//     PlcTask Outputs/Output.Out_Moter_Error <-> PlcTask Inputs/ExpConver.Out_Moter_Error
//     PlcTask Outputs/Output.Out_Moter_Running <-> PlcTask Inputs/ExpConver.Out_Moter_Running
//     PlcTask Outputs/Output.Out_Pos_sensor <-> PlcTask Inputs/ExpConver.Out_sensor
//     PlcTask Outputs/Output.PullOver_bBuzy <-> PlcTask Inputs/ExpConver.PullOver_bBuzy
//     PlcTask Outputs/Output.PullOver_bDone <-> PlcTask Inputs/ExpConver.PullOver_bDone
//     PlcTask Outputs/Output.PullOver_bError <-> PlcTask Inputs/ExpConver.PullOver_bError
//     PlcTask Outputs/Output.in_Pos_sensor <-> PlcTask Inputs/ExpConver.In_sensor

CONFIGURATION Main
    RESOURCE PLC ON TwinCAT3
        TASK PlcTask(INTERVAL := T#10ms, PRIORITY := 14);
        PROGRAM MAIN WITH PlcTask : MAIN;
    END_RESOURCE
END_CONFIGURATION

// ---- DUTs/ActionMode.TcDUT
{attribute 'qualified_only'}
{attribute 'strict'}
TYPE ActionMode :
(
	DoNothing	:= 0,
	AbsMove		:= 1,
	RelMove		:= 2,
	Home		:= 3,
	Find		:= 4
);
END_TYPE

// ---- DUTs/IO模組/IO_In16.TcDUT
TYPE IO_In16 :
STRUCT
	in AT %I* : ARRAY [1..16] OF BOOL;
END_STRUCT
END_TYPE

// ---- DUTs/IO模組/IO_Out16.TcDUT
TYPE IO_Out16 :
STRUCT
	Out AT %Q* : ARRAY [1..16] OF BOOL;
END_STRUCT
END_TYPE

// ---- DUTs/Jog_STRUCT/Jog_Laser_Group.TcDUT
TYPE Jog_Laser_Group :
STRUCT
	// 位置	
	Pos : XYZ_Point;
	
	// Jog模式 X軸 前進
	X_P_S : BOOL;
	// Jog模式 X軸 後退
	X_N_S : BOOL;
	
	// Jog模式 Y軸 前進
	Y_P_S : BOOL;
	// Jog模式 Y軸 後退
	Y_N_S : BOOL;
	
	// Jog模式 Z軸 前進
	Z_P_S : BOOL;
	// Jog模式 Z軸 後退
	Z_N_S : BOOL;

	// Jog模式 X軸 前進
	X_P : BOOL;
	// Jog模式 X軸 後退
	X_N : BOOL;
	
	// Jog模式 Y軸 前進
	Y_P : BOOL;
	// Jog模式 Y軸 後退
	Y_N : BOOL;
	
	// Jog模式 Z軸 前進
	Z_P : BOOL;
	// Jog模式 Z軸 後退
	Z_N : BOOL;
	
	
	// 雷射吹氣_狀態
	Laser_Blow_s : BOOL;
	// 雷射護蓋_狀態
	Laser_Cover_s : BOOL;
	

	// 雷射吹氣
	Laser_Blow : BOOL;
	// 雷射護蓋
	Laser_Cover : BOOL;
END_STRUCT
END_TYPE

// ---- DUTs/Jog_STRUCT/Jog_Fx_Group.TcDUT
TYPE Jog_Fx_Group :
STRUCT
	// 
	P_S : BOOL;
	// 後退
	N_S : BOOL;
	
	// 前進
	P : BOOL;
	// 後退
	N : BOOL;
	
	
	// 前進
	P_Fast_S : BOOL;
	// 後退
	N_Fast_S : BOOL;	

	// 前進
	P_Fast : BOOL;
	// 後退
	N_Fast : BOOL;
	
	
	// 下壓夾狀態
	V_Close_S : BOOL;
	// 下壓開狀態
	V_Open_S : BOOL;
	
	// 下壓夾
	V_Close : BOOL;
	// 下壓開
	V_Open : BOOL;
	
	// 滾輪夾狀態
	H_Close_S : BOOL;
	// 滾輪開狀態
	H_Open_S : BOOL;
	// 滾輪夾保持狀態
	H_Hold_S : BOOL;
	
	// 滾輪夾
	H_Close : BOOL;
	// 滾輪開
	H_Open : BOOL;
	// 滾輪夾保持
	H_Hold : BOOL;
	
	// 外部編碼器接觸
	ExEncTouch : BOOL;
	// 外部編碼器脫離
	ExEncExit : BOOL;
END_STRUCT
END_TYPE

// ---- DUTs/MachineState.TcDUT
{attribute 'qualified_only'}
{attribute 'strict'}
TYPE MachineState :
(
	standby := 0, 			// 待命
	Auto_mode := 2#01,		// 自動模式
	auto_mode_wait := 2#10,		// 自動模式等待中
	Remote_Auto_mode := 2#11,		// 遠端自動模式
	manual_mode := 2#100,	// 手動模式
	Homing_mode := 2#1000,		// 歸零模式
	
	error := 16#20,	// 發生錯誤
	Door := 16#40,		// 安全光柵觸發
	emergency := 16#80	// 緊急停止
) INT;
END_TYPE

// ---- DUTs/Sub_Step.TcDUT
TYPE Sub_Step :
STRUCT
	Step	: INT;
	
	bBuzy	: BOOL;
	bDone	: BOOL;
	bError	: BOOL;
END_STRUCT
END_TYPE

// ---- DUTs/TestAction.TcDUT
TYPE TestAction :
STRUCT
	// 選擇的動作 (1.軸移動、 2.等待完成、 3.等待時間 、4. 重複)
	ActionSelect: INT;
	
	// 選擇的軸 (動作1 有效)
	AxisSelect: INT;
	
	// 移動位置 (動作1 有效)
	Pos : REAL;
	
	// 移動速度 (動作1 有效)
	Speed: REAL;
	
	// 等待時間(動作3 有效)
	WaitTime : REAL;
	
	// 重複次數(動作4 有效)
	Cycles: UINT;
	
	// 重複動作(動作4 有效)
	Cycles_StartStep: UINT;
	
	// 重複次數(動作4 有效)
	Cycles_Done: UINT;
END_STRUCT
END_TYPE

// ---- DUTs/加工資料結構/材料加工資訊結構/tsSteelData.TcDUT
// 專案資料結構
TYPE tsSteelData :
STRUCT
	// 素材編號 (uuid)
	uid							: STRING(36);
	// 型鋼類型
	SteelType					: DINT;
	// 長度
	Length						: LREAL;
	// 高度
	Height						: LREAL;
	// 寬度
	Width						: LREAL;
	// 翼板厚度t1
	T1							: LREAL;
	// 翼板厚度t2
	T2							: LREAL;
	// 原點偏移
	OriginOffset				: LREAL;
	// 開啟預覽
	PreviewEnabled				: BOOL;
	// 預覽模式
	PreviewMode					: DINT;
	// 預覽時間
	PreviewTme					: DINT;
	// 「指定區域加工模式」的起始範圍
	rDesignateAreaRangeBegin	: LREAL;
	// 「指定區域加工模式」的結束範圍
	rDesignateAreaRangeEnd		: LREAL;
	
	// 上面的加工內容
	payloadTop					: STRING(36);
	// 下面的加工內容
	payloadBottom				: STRING(36);
	// 左面的加工內容
	payloadLeft					: STRING(36);
	// 右面的加工內容
	payloadRight				: STRING(36);
	
	// 全部加工完成
	bJobFinish					:BOOL;
END_STRUCT
END_TYPE

// ---- DUTs/加工資料結構/工單結構/WorkOrder_Data.TcDUT
// 專案資料結構
TYPE WorkOrder_Data :
STRUCT
	// 加工順序
	SN			: DINT;
	// 高
	Height		: LREAL;
	// 寬
	Width		: LREAL;
	// 素材編號 (uuid)
	steel_id	: STRING(36);
END_STRUCT
END_TYPE

// ---- DUTs/加工資料結構/雷射加工參數/LaserParameter_Data.TcDUT
TYPE LaserParameter_Data :
STRUCT
	// 加工參數代碼
	id				: DINT;
	// 螺徑(mm)
	SpiralDiameter	: LREAL;
	// 螺距(mm)
	SpiralDist		: LREAL;
	// 功率(%)
	Power			: DINT;
	// 速度(mm/S)
	Speed			: DINT;	
	// 頻率(KHZ)
	FREQ			: DINT;	
	// 脈波寬度(ns)
	PulseWidth		: DINT;	
END_STRUCT
END_TYPE

// ---- DUTs/加工資料結構/雷射加工資料/LaserProcess_Data.TcDUT
TYPE LaserProcess_Data :
// 115 byte
STRUCT
	// 資料的UID
	data_uid					: STRING(36);
	// 面的UID
	uid							: STRING(36);
	// 該面的序號(順序)
	paySerial					: DINT;
	// 使用雷射參數
	LaserParameter				: DINT;
	// 加工內容的x座標
	Point_X						: LREAL;
	// 加工內容的y座標
	Point_Y						: LREAL;
	// 加工內容的寬度
	Width						: LREAL;
	// 加工內容的高度
	Height						: LREAL;
	// 是否是QRCode
	isQRCode					: BOOL;
	// 已完成
	isDone						: BOOL;
	// QRCode字串
	qrcode_data					: STRING(100);
END_STRUCT
END_TYPE

// ---- DUTs/座標/XYZ_Point.TcDUT
TYPE XYZ_Point :
STRUCT
	X : LREAL;
	Y : LREAL;
	Z : LREAL;
END_STRUCT
END_TYPE

// ---- MSG/訊息格式/MsgLevel.TcDUT
{attribute 'qualified_only'}
{attribute 'strict'}
TYPE MsgLevel :
(
	Error	:= 4,
	Alarm	:= 2,
	Info	:= 1,
	None	:= 0
	
)INT;
END_TYPE

// ---- MSG/訊息格式/MsgStruct.TcDUT
{attribute 'pack_mode' := '1'} 
TYPE MsgStruct :
STRUCT
	// 訊息時間
	msgTIME		: DATE_AND_TIME;
	// 訊息等級
	Level		: MsgLevel;
	// 訊息號碼
	Number	: UINT;
	// 訊息附帶文字1
	MsgStr1	: WSTRING(80);
	// 訊息附帶文字2
	MsgStr2	: WSTRING(80);
	// 訊息全文
	raw_msg_str	: WSTRING(250);
END_STRUCT
END_TYPE

// ---- MSG/訊息格式/MsgStruct_RAW.TcDUT
{attribute 'pack_mode' := '1'} 
TYPE MsgStruct_RAW :
STRUCT
	// 訊息時間
	msgTIME		: DATE_AND_TIME;
	// 訊息等級
	Level		: MsgLevel;
	// 訊息號碼
	Number	: UINT;
	// 訊息附帶文字1
	MsgStr1	:  ARRAY[0..159] OF BYTE;
	// 訊息附帶文字2
	MsgStr2	: ARRAY[0..159] OF BYTE;
	// 訊息全文
	raw_msg_str	: ARRAY[0..499] OF BYTE;
END_STRUCT
END_TYPE

// ---- POUs/功能塊/資料庫 Postgre相關/相關結構/取得範圍內的加工資料/SQL_Get_Payload_Struct.TcDUT

TYPE SQL_Get_Payload_Struct :
STRUCT
	// 
	Payload_Uid : STRING(36);
	PosBegain	: LREAL;
	PosEnd	: LREAL;
END_STRUCT
END_TYPE

// ---- POUs/功能塊/資料庫 Postgre相關/相關結構/取得X點/SQL_GetPosX_Struct.TcDUT
// 取得檔案的參數
TYPE SQL_GetPosX_Struct :
STRUCT
	Payload_A_Uid : STRING(36);
	Payload_B_Uid : STRING(36);
	Payload_C_Uid : STRING(36);
	Payload_D_Uid : STRING(36);
	Pos	: LREAL;
END_STRUCT
END_TYPE

// ---- POUs/功能塊/資料庫 Postgre相關/相關結構/寫入起始時間/Payload_Write_Time.TcDUT
TYPE Payload_Write_Time :
STRUCT
	// 時間
	Start_TIME		: DATE_AND_TIME;
	// 目標uid
	Uid : STRING(36);
END_STRUCT
END_TYPE

// ---- POUs/功能塊/資料庫 Postgre相關/記錄用/程式紀錄/StepLog_Struct.TcDUT
TYPE StepLog_Struct :
STRUCT
	step_number : DINT;
	created_at : LINT;
	program_name : STRING(80);
	extras_Srt : STRING(255) := '{}';
END_STRUCT
END_TYPE

// ---- POUs/動作流程控制/測試功能/Sql_TestData.TcDUT
TYPE Sql_TestData :
STRUCT
	ID : LINT;
	LogTime : DATE_AND_TIME;
	
END_STRUCT
END_TYPE

// ---- POUs/動作流程控制/測試功能/Sql_TestWriteData.TcDUT
TYPE Sql_TestWriteData :
STRUCT
	LogTime : DATE_AND_TIME;
END_STRUCT
END_TYPE

// ---- GVLs/Axis.TcGVL
{attribute 'TcContextName':='PlcTask'}
VAR_GLOBAL
// 軸控制
// ============== 滾輪軸 ==============
	//  前
	Axis_FX1: AXIS_REF;
	//  後
	Axis_FX2: AXIS_REF;
	
	Fx : AxisFx;
	
	
// ============== A ==============
	
	// X軸
	Axis_AX: AXIS_REF;
	
	// Y軸
	Axis_AY: AXIS_REF;
	// Z軸
	Axis_AZ1: AXIS_REF;
	Axis_AZ2: AXIS_REF;
	
	GaX : AxisBase;
	GaY : AxisBase;
	GaZ : MultipleAxisBase;
	

	
// ============== B ==============
	// X軸
	Axis_BX: AXIS_REF;
	// Y軸
	Axis_BY1: AXIS_REF;
	Axis_BY2: AXIS_REF;
	// Z軸
	Axis_BZ: AXIS_REF;
	
	GbX : AxisBase;
	GbY : MultipleAxisBase;
	GbZ : AxisBase;
	
// ============== C ==============
	// X軸
	Axis_CX: AXIS_REF;
	// Y軸
	Axis_CY: AXIS_REF;
	// Z軸
	Axis_CZ1: AXIS_REF;
	Axis_CZ2: AXIS_REF;
	
	GcX : AxisBase;
	GcY : AxisBase;
	GcZ : MultipleAxisBase;
	
// ============== D ==============
	// X軸
	Axis_DX: AXIS_REF;
	// Y軸
	Axis_DY: AXIS_REF;
	// Z軸
	Axis_DZ: AXIS_REF;
	
	GdX : AxisBase;
	GdY : AxisBase;
	GdZ : AxisBase;


//  ============== 整體軸速度 ==============	
	Override: LREAL := 100;
	bIsHome: BOOL;
	bPower: BOOL;
	
{region "============= 編碼器  ============="}
	Encoder_FxA_PosEnc	:	MDP5001_511_5ED3066D;
	Encoder_FxB_PosEnc	:	MDP5001_511_5ED3066D;
		 
	Encoder_FxA_Clamp	:	MDP5001_511_5ED3066D;
	Encoder_FxB_Clamp	:	MDP5001_511_5ED3066D;
		 
	Encoder_FxA_ExPosEnc	:	MDP5001_511_5ED3066D;
	Encoder_FxB_ExPosEnc	:	MDP5001_511_5ED3066D;
	
	// FxA外部位置
	FxA_Exp_Pos				: LREAL;
	// FxB外部位置
	FxB_Exp_Pos				: LREAL;
	
	// Fx整合位置
	Fx_Exp_Pos				: LREAL;
{endregion}
	

	id: INT;
	
	
END_VAR


VAR_GLOBAL PERSISTENT
	// Gax軸 移動距離
	GaX_total_Move: LREAL;
	// Gay軸 移動距離
	GaY_total_Move: LREAL;
	// Gaz軸 移動距離
	GaZ_total_Move: LREAL;
	
	// Gax軸 移動距離
	GbX_total_Move: LREAL;
	// Gay軸 移動距離
	GbY_total_Move: LREAL;
	// Gaz軸 移動距離
	GbZ_total_Move: LREAL;
	
	// Gax軸 移動距離
	GcX_total_Move: LREAL;
	// Gay軸 移動距離
	GcY_total_Move: LREAL;
	// Gaz軸 移動距離
	GcZ_total_Move: LREAL;
	
	// Gax軸 移動距離
	GdX_total_Move: LREAL;
	// Gay軸 移動距離
	GdY_total_Move: LREAL;
	// Gaz軸 移動距離
	GdZ_total_Move: LREAL;
	
	// Gax軸 移動距離
	GaX_Last_Oil: LREAL;
	// Gay軸 移動距離
	GaY_Last_Oil: LREAL;
	// Gaz軸 移動距離
	GaZ_Last_Oil: LREAL;
	
	// Gax軸 移動距離
	GbX_Last_Oil: LREAL;
	// Gay軸 移動距離
	GbY_Last_Oil: LREAL;
	// Gaz軸 移動距離
	GbZ_Last_Oil: LREAL;
	
	// Gax軸 移動距離
	GcX_Last_Oil: LREAL;
	// Gay軸 移動距離
	GcY_Last_Oil: LREAL;
	// Gaz軸 移動距離
	GcZ_Last_Oil: LREAL;
	
	// Gax軸 移動距離
	GdX_Last_Oil: LREAL;
	// Gay軸 移動距離
	GdY_Last_Oil: LREAL;
	// Gaz軸 移動距離
	GdZ_Last_Oil: LREAL;
END_VAR

// ---- GVLs/GrobelVariable.TcGVL
VAR_GLOBAL
// 雜項
	
	ProgramReset:BOOL;
	
	// 機器已回零
	bHome : BOOL;
	
	// 
	LogFx : FxErrPos;
END_VAR

VAR_GLOBAL PERSISTENT
	// 運轉次數
	uRunCounter:UDINT;
END_VAR

// ---- GVLs/Hmi.TcGVL
{attribute 'qualified_only'}
VAR_GLOBAL
(* ================= 模式選擇 ================= *)
	// 自動模式
	Auto_Mode : BOOL;

	// Jog模式
	Jog_Mode : BOOL;
	
	// 手輪模式
	MPG_Mode : BOOL;
	
	// 選擇的模式
	Mode_Select : DINT;

(* ================= 自動模式 ================= *)
	// 自動流程 開始執行
	Auto_Start : BOOL;
	
	// 一循環流程 開始執行
	Auto_OneCycle_Start : BOOL;
	
	// 自動流程 暫停/繼續
	Auto_Pause:BOOL;
	
	// 自動流程 加工單
	Auto_ProjectWorkOrder_uuid : STRING;

	// 自動流程 動作選擇
	Auto_ProgramSelect : DINT;

	// 自動流程 動作執行中
	Auto_bBuzy : BOOL;
	
	// 自動流程 動作完成
	Auto_bDone : BOOL;
	
	

	// 動作狀態通知
	ActinoNow:WSTRING;
	

	// 狀態欄 機器動作中
	State: MachineState := MACHINESTATE.standby;
	
	
(*==================== Jog模式====================*)
	// Jog模式 軸組選擇
	Jog_GroupSelect : DINT;
	
	// Jog模式 互鎖解除
	Jog_UnLimite : BOOL;
	
	// Jog模式 速度
	Jog_Speed: REAL := 30;
	
	
	
	Jog_move_to : LREAL;
	Jog_move_to_start : BOOL;
	Jog_move_to_bBuzy : BOOL;
	Jog_move_to_bDone : BOOL;
	
	// JOG 設定動作群組
	Jog_Set_GroupA: BOOL;
	Jog_Set_GroupB: BOOL;
	Jog_Set_GroupC: BOOL;
	Jog_Set_GroupD: BOOL;
	
	// Jog模式 X軸 前進
	Jog_X_P : BOOL;
	// Jog模式 X軸 後退
	Jog_X_N : BOOL;
	
	// Jog模式 Y軸 前進
	Jog_Y_P : BOOL;
	// Jog模式 Y軸 後退
	Jog_Y_N : BOOL;
	
	// Jog模式 Z軸 前進
	Jog_Z_P : BOOL;
	// Jog模式 Z軸 後退
	Jog_Z_N : BOOL;
	
	
(*==================== 原點設置 ====================*)
	// 設定 X軸 原點
	Set_X_Home : BOOL;
	// 設定 X軸 正極限
	Set_X_P_Limite : BOOL;
	// 設定 Y軸 原點
	Set_Y_Home : BOOL;
	// 設定 Y軸 正極限
	Set_Y_P_Limite : BOOL;
	// 設定 Z軸 原點
	Set_Z_Home : BOOL;
	// 設定 Z軸 正極限
	Set_Z_P_Limite : BOOL;

	
	
	// 將極限設定 參數 寫入軸
	Set_Axis_Limit : BOOL;
	
	// 錯誤重置
	SysErrorRest: BOOL;
	


	
	
END_VAR

// ---- GVLs/Hmi_Web.TcGVL
{attribute 'qualified_only'}
VAR_GLOBAL
(* ================= 模式選擇 ================= *)
	// 人機 > PLC WatchDog
	Watchdog_in : BOOL;
	
	// PLC > 人機 WatchDog
	Watchdog_Out : BOOL;
	
	// 錯誤重置
	SysErrorRest: BOOL;
	
	// 自動模式
	Auto_Mode : BOOL;
	
	// 單步模式
	Auto_Step_mode_Enable :BOOL;
	
	
	// 單步模式生效
	Auto_Step_active :BOOL;

	// Jog模式
	Jog_Mode : BOOL;
	
	// 手輪模式
	MPG_Mode : BOOL;
	
	// 選擇的模式
	Mode_Select : DINT;
	

(* ================= 自動模式 ================= *)
	// 自動流程 開始的專案UUID
	Auto_ProjectWorkOrder_uuid : STRING(36);
	// 自動流程 開始的專案UUID
	Start_WorkOrder_UUID : STRING(36);

	// 自動流程 開始執行
	Auto_Start : BOOL;
	
	Auto_OneCycle_Start : BOOL;
	
	
	
	

	
	// 自動流程 暫停/繼續
	Auto_Pause:BOOL;

	// 自動流程 動作選擇
	Auto_ProgramSelect : DINT;

	// 自動流程 動作執行中
	Auto_bBuzy : BOOL;
	
	// 自動流程 動作完成
	Auto_bDone : BOOL;
	
	// 自動流程 原點復歸
	Auto_homming : BOOL;
	
	// 動作狀態通知
	ActinoNow:WSTRING;
	
	// 狀態欄 機器動作中
	State: MachineState := MACHINESTATE.standby;
	
	
	// 雷射A 控制
	Process_Data_UUID_A				: STRING(36);
 	Process_Data_UUID_A_Start		: BOOL;
	// 雷射B 控制
	Process_Data_UUID_B				: STRING(36);
 	Process_Data_UUID_B_Start		: BOOL;
	// 雷射C 控制
	Process_Data_UUID_C				: STRING(36);
 	Process_Data_UUID_C_Start		: BOOL;
	// 雷射D 控制
	Process_Data_UUID_D				: STRING(36);
 	Process_Data_UUID_D_Start		: BOOL;
	
(*==================== Jog模式====================*)
	// Jog模式 軸組選擇
	Jog_GroupSelect : DINT;
	
	// Jog模式 互鎖解除
	Jog_UnLimite : BOOL;
	
	// Jog模式 速度
	Jog_Speed: REAL := 80;
	
	jog_trig_R : ARRAY [0..9] OF R_TRIG;


	jog_trig_F : ARRAY [0..9] OF F_TRIG; 
	
	
(*==================== Ga Jog模式====================*)	
	// Jog模式Ga X軸 前進
	Jog_Ga : Jog_Laser_Group;
	

(*==================== Gb Jog模式====================*)	
	// Jog模式Gb X軸 前進
	Jog_Gb : Jog_Laser_Group;

(*==================== Gc Jog模式====================*)	
	// Jog模式Gc
	Jog_Gc : Jog_Laser_Group;

(*==================== Gd Jog模式====================*)	
	// Jog模式Gd
	Jog_Gd : Jog_Laser_Group;
	
(*==================== FX A Jog模式====================*)	
	// Jog模式FxA
	Jog_FxA : Jog_Fx_Group;
	
(*==================== FX A Jog模式====================*)	
	// Jog模式FxB
	Jog_FxB : Jog_Fx_Group;
	
	// 油壓幫浦
	Oil_Pump:BOOL;
(*==================== Fx 目前位置====================*)	
	Fx_Pos			:LREAL;		// Fx 馬達位置
	FxA_Ex_Pos		:LREAL;		// FxA 測長盤
	FxB_Ex_Pos		:LREAL;		// FxB 測長盤

	FxA_H_Pos		:LREAL;		// FxA 油壓夾輪位置
	FxB_H_Pos		:LREAL;		// FxB 油壓夾輪位置
	
	
(*==================== Ga 工件座標系位置====================*)	
	WCS_A : XYZ_Point;
(*==================== Gb 工件座標系位置====================*)	
	WCS_B : XYZ_Point;
(*==================== Gc 工件座標系位置====================*)	
	WCS_C : XYZ_Point;
(*==================== Gd 工件座標系位置====================*)	
	WCS_D : XYZ_Point;
	
	
END_VAR
VAR_GLOBAL PERSISTENT
	// 工件誤差修正
	Auto_Steel_X_Offset : LREAL;
END_VAR

// ---- GVLs/MaCfg.TcGVL
{attribute 'qualified_only'}
VAR_GLOBAL PERSISTENT
	(* ======= Group A =======*)
	// 雷射頭A焦距
	laserA_Dis : REAL := 297;
	// 軸組A的 雷射測距可以測得範圍
	laserA_Y_DisSensorArrivePos	:REAL := 300;
	// 軸組Ax的 雷射測距點 到 雷射頭的中心點
	laserA_X_DisSensor2LaserCenter : REAL := -76;
	// 軸組Ay的 雷射測距點 到 雷射頭的中心點
	laserA_Y_DisSensor2LaserCenter : REAL := 12;
	// 軸組A的 Y 基準位置 (實際無法到達) (搭配 FindY 指令，可以測得工件高度)
	laserA_Y_ReferencePos : REAL := 677.7;
	
	(* ======= Group B =======*)
	// 雷射頭B焦距
	laserB_Dis	: REAL := 297;
	// 軸組B的 雷射測距可以測得範圍
	laserB_Y_DisSensorArrivePos		: REAL := 185;
	
	// 軸組Bx的 雷射測距點 到 雷射頭的中心點
	laserB_X_DisSensor2LaserCenter	: REAL := -0.6;
	// 軸組By的 雷射測距點 到 雷射頭的中心點
	laserB_Y_DisSensor2LaserCenter	: REAL := -77.2;
	
	// 軸組B的 Y 基準位置 (搭配 FindY 指令，可以測得工件高度)
	laserB_Y_ReferencePos	: REAL := 1344.5599;
	// 軸組B的 Z 基準位置 (實際無法到達)
	laserB_Z_ReferencePos	: REAL := -298;
	
	// 軸組Bx的 雷射測距點 到 雷射頭的中心點
	laserB_Y_safetyPos	: REAL := 20;
	// 軸組B的Z軸的安全位置
	laserB_Z_safetyPos		: REAL := 500;
	
	
	(* ======= Group C =======*)
	// 雷射頭C焦距
	laserC_Dis : REAL := 298;
	// 軸組C的 雷射測距可以測得範圍
	laserC_Y_DisSensorArrivePos	:REAL := 185;
	// 軸組Cx的 雷射測距點 到 雷射頭的中心點
	laserC_X_DisSensor2LaserCenter : REAL := 77.9;
	// 軸組Cy的 雷射測距點 到 雷射頭的中心點
	laserC_Y_DisSensor2LaserCenter : REAL := 5.8;
	// 軸組C的 Y 基準位置 (實際無法到達) (搭配 FindY 指令，可以測得工件高度)
	laserC_Y_ReferencePos : REAL := 605.3;
	// 軸組C的 Z 基準位置 (實際無法到達)
	laserC_Z_ReferencePos : REAL := -416;
	
	(* ======= Group D =======*)
	// 雷射頭D焦距
	laserD_Dis : REAL := 299;
	// 軸組D的 雷射測距可以測得範圍
	laserD_Y_DisSensorArrivePos	:REAL := 185;
	// 軸組D的 雷射測距點 到 雷射頭的中心點
	laserD_Y_DisSensor2LaserDenter : REAL := 3.1;
	// 軸組D的 Y 基準位置 (實際無法到達) (搭配 FindY 指令，可以測得工件高度)
	laserD_Y_ReferencePos : REAL := 1286.064821;
	
	
	// FxB被動編碼器 比例(mm/plus)
	FxA_Enc_Scale : LREAL := 0.046047445;
	// FxB測常盤編碼器 比例(mm/plus)
	FxA_Enc_Ext_Scale : LREAL := 0.14459929225;
	
	// FxB被動編碼器 比例(mm/plus)
	FxB_Enc_Scale : LREAL := 0.046047445;
	// FxB測常盤編碼器 比例(mm/plus)
	FxB_Enc_Ext_Scale : LREAL := 0.14459929225;
	
	
	
	// 進料端反轉
	bInSite_Invert: BOOL;
	
	//
	// AC夾輪的零點位置 ( 空夾位置 + 空夾兩夾輪間距(70))
	FxA_Clamp_Zero_Pos: LREAL := 1297.4;
	// BD夾輪的零點位置 ( 空夾位置 + 空夾兩夾輪間距(70))
	FxB_Clamp_Zero_Pos: LREAL := 1296.49;
	
	// 雷射動作超時
	LaserPrinter_Timeout : DINT := 60000;
	
END_VAR

// ---- GVLs/IO.TcGVL
{attribute 'qualified_only'}
{attribute 'TcContextName':='PlcTask'}
VAR_GLOBAL
{region "============= EL1409_1 ============="}
	// 緊急停止-PB
	i101 AT %I*: BOOL;
	// IPC開機-PB
	i102 AT %I*: BOOL;
	// 程式暫停-PB
	i103 AT %I*: BOOL;
	// 程式啟動-PB
	i104 AT %I*: BOOL;
	// 重置-PB
	i105 AT %I*: BOOL;
	// 原點模式A-KS
	i106 AT %I*: BOOL;
	// 原點模式B-KS
	i107 AT %I*: BOOL;
	// 吋動-KS
	i108 AT %I*: BOOL;
	// 半自動-KS
	i109 AT %I*: BOOL;
	// 全自動-KS
	i110 AT %I*: BOOL;
	// 門解鎖-KS
	i111 AT %I*: BOOL;
	// 安全模組重置-PB
	i112 AT %I*: BOOL;
	// 模式選擇A-KS
	i113 AT %I*: BOOL;
	// 模式選擇B-KS
	i114 AT %I*: BOOL;
	// 雷射D鏡頭防護蓋開-PB
	i115 AT %I*: BOOL;
	// 雷射D鏡頭防護蓋關-PB
	i116 AT %I*: BOOL;
 {endregion}
{region "============= EL1409_2 ============="}
	// 吋動 X+
	i201 AT %I*: BOOL;
	// 吋動 X-
	i202 AT %I*: BOOL;
	// 吋動 Y+
	i203 AT %I*: BOOL;
	// 吋動 Y-
	i204 AT %I*: BOOL;
	// 吋動 Z+_PB
	i205 AT %I*: BOOL;
	// 吋動 Z-_PB
	i206 AT %I*: BOOL;
	// 螢幕旋轉
	i207 AT %I*: BOOL;
	// 油壓啟動
	i208 AT %I*: BOOL;
	// 油壓馬達過負載
	i209 AT %I*: BOOL;
	// 油壓散熱循環馬達過負載
	i210 AT %I*: BOOL;
	// 安全模組信號
	i211 AT %I*: BOOL;
	// 氣壓壓力檢知
	i212 AT %I*: BOOL;
	// 雷射A遮蔽信號
	i213 AT %I*: BOOL;
	// 雷射B遮蔽信號
	i214 AT %I*: BOOL;
	// 雷射C遮蔽信號
	i215 AT %I*: BOOL;
	// 雷射D遮蔽信號
	i216 AT %I*: BOOL;
{endregion}
{region "============= EL1409_3 ============="}
	// 潤滑油A液位檢知
	i301 AT %I*: BOOL;
	// 潤滑油A壓力檢知
	i302 AT %I*: BOOL;
	// Ax 正極限-LS
	i303 AT %I*: BOOL;
	// Ax 負極限-LS
	i304 AT %I*: BOOL;
	// Ay 正極限-LS
	i305 AT %I*: BOOL;
	// Ay 負極限-LS
	i306 AT %I*: BOOL;
	// Az 正極限-LS
	i307 AT %I*: BOOL;
	// Az 負極限-LS
	i308 AT %I*: BOOL;
	// 潤滑油D液位檢知
	i309 AT %I*: BOOL;
	// 潤滑油D壓力檢知
	i310 AT %I*: BOOL;
	// Dx 正極限
	i311 AT %I*: BOOL;
	// Dx 負極限
	i312 AT %I*: BOOL;
	// Dy 正極限
	i313 AT %I*: BOOL;
	// Dy 負極限
	i314 AT %I*: BOOL;
	// Dz 正極限
	i315 AT %I*: BOOL;
	// Dz 負極限
	i316 AT %I*: BOOL;
 {endregion}
{region "============= EL1409_4 ============="}
	// 潤滑油B液位檢知
	i401 AT %I*: BOOL;
	// 潤滑油B壓力檢知
	i402 AT %I*: BOOL;
	// Bx 正極限-LS
	i403 AT %I*: BOOL;
	// Bx 負極限-LS
	i404 AT %I*: BOOL;
	// Bz 正極限-LS
	i405 AT %I*: BOOL;
	// Bz 負極限-LS
	i406 AT %I*: BOOL;
	// AB區雷射極限開關-LS
	i407 AT %I*: BOOL;
	// BC區雷射極限開關-LS
	i408 AT %I*: BOOL;
	// 潤滑油C液位檢知
	i409 AT %I*: BOOL;
	// 潤滑油C壓力檢知
	i410 AT %I*: BOOL;
	// Cx 正極限-LS
	i411 AT %I*: BOOL;
	// Cx 負極限-LS
	i412 AT %I*: BOOL;
	// Cy 正極限-LS
	i413 AT %I*: BOOL;
	// Cy 負極限-LS
	i414 AT %I*: BOOL;
	// Cz 正極限
	i415 AT %I*: BOOL;
	// 
	i416 AT %I*: BOOL;
 {endregion}
{region "============= EL1409_5 ============="}
	// 下壓A原點
	i501 AT %I*: BOOL;
	// 下壓B原點
	i502 AT %I*: BOOL;
	// 下壓C原點
	i503 AT %I*: BOOL;
	// 下壓D原點
	i504 AT %I*: BOOL;
	// 下壓A壓力到達
	i505 AT %I*: BOOL;
	// 下壓B壓力到達
	i506 AT %I*: BOOL;
	// 下壓C壓力到達
	i507 AT %I*: BOOL;
	// 下壓D壓力到達
	i508 AT %I*: BOOL;
	// 側壓原點(AC)
	i509 AT %I*: BOOL;
	// 側壓原點(BD)
	i510 AT %I*: BOOL;
	// 材料原點偵測
	i511 AT %I*: BOOL;
	// 材料脫離點
	i512 AT %I*: BOOL;
	// 材料整料點
	i513 AT %I*: BOOL;
	// 鏡頭蓋 關
	i514 AT %I*: BOOL;
	// 鏡頭蓋 開
	i515 AT %I*: BOOL;
	// 
	i516 AT %I*: BOOL;
 {endregion}
{region "============= EL1409_6 ============="}
	// 手輪軸向X
	i601 AT %I*: BOOL;
	// 手輪軸向Y
	i602 AT %I*: BOOL;
	// 手輪軸向Z
	i603 AT %I*: BOOL;
	// 手輪倍率
	i604 AT %I*: BOOL;
	// 手輪倍率
	i605 AT %I*: BOOL;
	// 手輪區域選擇A
	i606 AT %I*: BOOL;
	// 手輪區域選擇B
	i607 AT %I*: BOOL;
	// 手輪區域選擇C
	i608 AT %I*: BOOL;
	// 手輪區域選擇D
	i609 AT %I*: BOOL;
	// 手輪急停
	i610 AT %I*: BOOL;
	// 手輪始能
	i611 AT %I*: BOOL;
	// 預留
	i612 AT %I*: BOOL;
	// 預留
	i613 AT %I*: BOOL;
	// 預留
	i614 AT %I*: BOOL;
	// 預留
	i615 AT %I*: BOOL;
	// 預留
	i616 AT %I*: BOOL;
{endregion}
{region "============= Murr IMPACT67 ============="}
	// X0.4
	i701 AT %I*: BOOL;
	// X0.2
	i702 AT %I*: BOOL;
	// X1.4
	i703 AT %I*: BOOL;
	// X1.2
	i704 AT %I*: BOOL;
	// X2.4
	i705 AT %I*: BOOL;
	// X2.2
	i706 AT %I*: BOOL;
	// X3.4
	i707 AT %I*: BOOL;
	// X3.2
	i708 AT %I*: BOOL;
	// X4.4 工件感應器 出口
	i709 AT %I*: BOOL;
	// X4.2 工件原點 (下)
	i710 AT %I*: BOOL;
	// X5.4 工件感應器 入口
	i711 AT %I*: BOOL;
	// X5.2
	i712 AT %I*: BOOL;
	// X6.4 工件原點 (AC夾輪)
	i713 AT %I*: BOOL;
	// X6.2
	i714 AT %I*: BOOL;
	// X7.4
	i715 AT %I*: BOOL;
	// X7.2
	i716 AT %I*: BOOL;
{endregion}	
	
{region "============= EL2409_7 ============="}
	// IPC啟動指示燈 
	q101 AT %Q*: BOOL;
	// 程式暫停指示燈
	q102 AT %Q*: BOOL;
	// 程式啟動指示燈
	q103 AT %Q*: BOOL;
	// 重置指示燈
	q104 AT %Q*: BOOL;
	// 原點完成指示燈A
	q105 AT %Q*: BOOL;
	// 原點完成指示燈B(門開關)
	q106 AT %Q*: BOOL;
	// 吋動模式指示燈
	q107 AT %Q*: BOOL;
	// 半自動模式指示燈
	q108 AT %Q*: BOOL;
	// 全自動模式指示燈
	q109 AT %Q*: BOOL;
	// 安全門解鎖
	q110 AT %Q*: BOOL;
	// 安全模組腹歸指示燈
	q111 AT %Q*: BOOL;
	// 日光燈開/關
	q112 AT %Q*: BOOL;
	// 警示燈 綠燈
	q113 AT %Q*: BOOL;
	// 警示燈 黃燈
	q114 AT %Q*: BOOL;
	// 警示燈 紅燈
	q115 AT %Q*: BOOL;
	// 警示燈 Bz
	q116 AT %Q*: BOOL;
{endregion}
{region "============= EL2409_8 ============="}
	// IPC啟動輸出
	q201 AT %Q*: BOOL;
	// 主機油壓馬達啟動
	q202 AT %Q*: BOOL;
	// 主機油壓高壓閥啟動
	q203 AT %Q*: BOOL;
	// A潤滑油啟動運轉
	q204 AT %Q*: BOOL;
	// B潤滑油啟動運轉
	q205 AT %Q*: BOOL;
	// C潤滑油啟動運轉
	q206 AT %Q*: BOOL;
	// D潤滑油啟動運轉
	q207 AT %Q*: BOOL;
	// 下壓A區上升
	q208 AT %Q*: BOOL;
	// 下壓A區下降
	q209 AT %Q*: BOOL;
	// 下壓B區上升
	q210 AT %Q*: BOOL;
	// 下壓B區下降
	q211 AT %Q*: BOOL;
	// 下壓C區上升
	q212 AT %Q*: BOOL;
	// 下壓C區下降
	q213 AT %Q*: BOOL;
	// 下壓D區上升
	q214 AT %Q*: BOOL;
	// 下壓D區下降
	q215 AT %Q*: BOOL;
	// 主機油壓低壓閥啟動
	q216 AT %Q*: BOOL;
{endregion}
{region "============= EL2409_9 ============="}
	// 側壓AC前進夾緊
	q301 AT %Q*: BOOL;
	// 側壓AC後退放鬆
	q302 AT %Q*: BOOL;
	// 側壓BD前進夾緊
	q303 AT %Q*: BOOL;
	// 側壓BD後退放鬆
	q304 AT %Q*: BOOL;
	// 雷射A吹氣
	q305 AT %Q*: BOOL;
	// 雷射B吹氣
	q306 AT %Q*: BOOL;
	// 雷射C吹氣
	q307 AT %Q*: BOOL;
	// 雷射D吹氣
	q308 AT %Q*: BOOL;
	// 雷射D保護蓋開
	q309 AT %Q*: BOOL;
	// 雷射D保護蓋關
	q310 AT %Q*: BOOL;
	// A側 外部編碼器 進
	q311 AT %Q*: BOOL;
	// A側 外部編碼器 退
	q312 AT %Q*: BOOL;
	// B側 外部編碼器 進
	q313 AT %Q*: BOOL;
	// B側 外部編碼器 退
	q314 AT %Q*: BOOL;
	// 預留
	q315 AT %Q*: BOOL;
	// 預留
	q316 AT %Q*: BOOL;
{endregion}
	
END_VAR

// ---- GVLs/PosC.TcGVL
{attribute 'qualified_only'}
VAR_GLOBAL PERSISTENT
	
	// 設定 A區X軸 正極限
	GaX_P_Limite : REAL;
	// 設定 A區X軸 負極限
	GaX_N_Limite : REAL;
	// 設定 A區Y軸 正極限
	GaY_P_Limite : REAL;
	// 設定 A區Y軸 負極限
	GaY_N_Limite : REAL;
	// 設定 A區Z軸 正極限
	GaZ_P_Limite : REAL;
	// 設定 A區Z軸 負極限
	GaZ_N_Limite : REAL;
	
	// 設定 A區Z軸 兩軸差
	GaZ_Diff :REAL;
	
	// GaX待機位置
	pos_GaX_stanby : REAL;
	// GaY待機位置
	pos_GaY_stanby : REAL;
	// GaZ待機位置
	pos_GaZ_stanby : REAL;
	
	// 設定 B區X軸 正極限
	GbX_P_Limite : REAL;
	// 設定 B區X軸 負極限
	GbX_N_Limite : REAL;
	// 設定 B區Y軸 正極限
	GbY_P_Limite : REAL;
	// 設定 B區Y軸 負極限
	GbY_N_Limite : REAL;
	// 設定 B區Z軸 正極限
	GbZ_P_Limite : REAL;
	// 設定 B區Z軸 負極限
	GbZ_N_Limite : REAL;
	
	// 設定 B區Y軸 兩軸差
	GbY_Diff :REAL;
	
	// GbX待機位置
	pos_GbX_stanby : REAL;
	// GbY待機位置
	pos_GbY_stanby : REAL;
	// GbZ待機位置
	pos_GbZ_stanby : REAL;
	
	// 設定 C區X軸 正極限
	GcX_P_Limite : REAL;
	// 設定 C區X軸 負極限
	GcX_N_Limite : REAL;
	// 設定 C區Y軸 正極限
	GcY_P_Limite : REAL;
	// 設定 C區Y軸 負極限
	GcY_N_Limite : REAL;
	// 設定 C區Z軸 正極限
	GcZ_P_Limite : REAL;
	// 設定 C區Z軸 負極限
	GcZ_N_Limite : REAL;
	
	// 設定 C區Z軸 兩軸差
	GcZ_Diff :REAL;
	
	// GcX待機位置
	pos_GcX_stanby : REAL;
	// GcY待機位置
	pos_GcY_stanby : REAL;
	// GcZ待機位置
	pos_GcZ_stanby : REAL;
	
	// 設定 D區X軸 正極限
	GdX_P_Limite : REAL;
	// 設定 D區X軸 負極限
	GdX_N_Limite : REAL;
	// 設定 D區Y軸 正極限
	GdY_P_Limite : REAL;
	// 設定 D區Y軸 負極限
	GdY_N_Limite : REAL;
	// 設定 D區Z軸 正極限
	GdZ_P_Limite : REAL;
	// 設定 D區Z軸 負極限
	GdZ_N_Limite : REAL;
	
	// GdX待機位置
	pos_GdX_stanby : REAL;
	// GdY待機位置
	pos_GdY_stanby : REAL;
	// GdZ待機位置
	pos_GdZ_stanby : REAL;
	
	Fx_HomeOffset : REAL;
END_VAR

// ---- GVLs/ProjectData.TcGVL
{attribute 'qualified_only'}
VAR_GLOBAL
	// 使用的料
	WorkOrder_Now : WorkOrder_Data;
	
	// 在自動料架上 料的數量
	WorkOrder_Num_On_Wait : INT;
	
	// 狀態為 inSide(入料) 的料
	WorkOrder_inSide 	: WorkOrder_Data;
	// 狀態為 alignment(無靠邊插單) 的料
	WorkOrder_alignment 	: WorkOrder_Data;
	// 狀態為 inserts(插單) 的料
	WorkOrder_inserts 	: WorkOrder_Data;
	
	
	Now_Steel	: tsSteelData;
	old_Steel	: tsSteelData;
	
	// 接縫 (出現在BH，板長不夠時兩塊板連接的位置)
	Joint_Pos : LREAL := 0;
	
	Now_Steel_H_m : LREAL;
	Now_Steel_W_m : LREAL;
	
	// 雷射參數 暫存區
	LaserParameter : ARRAY [0..3] OF LaserParameter_Data;
	

	// A面加工資訊數量
	Now_Steel_Payload_A_DataNumber : INT;
	// A面加工資訊
	Payload_A_Data_Now : LaserProcess_Data;
	// A面加工資訊預讀
	Payload_A_Data_buff : ARRAY [0..50] OF LaserProcess_Data;
	// A面加工完成數量
	Now_Steel_Payload_A_DataNumber_Done : INT;
	
	
	// B面加工資訊數量
	Now_Steel_Payload_B_DataNumber : INT;
	// B面加工資訊
	Payload_B_Data_Now : LaserProcess_Data; //115 byte
	// B面加工資訊緩衝區
	Payload_B_Data_buff : ARRAY [0..50] OF LaserProcess_Data;
	// B面加工完成數量
	Now_Steel_Payload_B_DataNumberDone : INT;
	
	
	// C面加工資訊數量
	Now_Steel_Payload_C_DataNumber : INT;
	// C面加工資訊
	Payload_C_Data_Now : LaserProcess_Data; //115 byte
	// C面加工資訊緩衝區
	Payload_C_Data_buff : ARRAY [0..50] OF LaserProcess_Data;
	// C面加工完成數量
	Now_Steel_Payload_C_DataNumberDone : INT;
	
	
	// D面加工資訊數量
	Now_Steel_Payload_D_DataNumber : INT;
	// D面加工資訊
	Payload_D_Data_Now : LaserProcess_Data; //115 byte
	// D面加工資訊緩衝區
	Payload_D_Data_buff : ARRAY [0..50] OF LaserProcess_Data;
	// D面加工完成數量
	Now_Steel_Payload_D_DataNumberDone : INT;
	
	
END_VAR

// ---- GVLs/Safety.TcGVL

VAR_GLOBAL
	// 緊急停止
	Estop: BOOL;	
	// 光柵
	Door: BOOL;
	
	SystemError :BOOL;
	
	SystemAlarm :BOOL;
	
	
	close_Air_Pressure_Check:bool;
	
	//關閉前方光柵
	close_Door_Bad:BOOL;
	//關閉臺車出入口光柵
	close_Door_Car_Gate:BOOL;
	//關閉臺車周圍光柵
	close_Door_Car_Around:BOOL;
	
	//關閉鏈條斷裂檢
	close_Chain_Break_Check: BOOL;
	
	// 真空壓力感應器
	VacuumSensor: BOOL;
END_VAR

// ---- GVLs/SensorTest.TcGVL
{attribute 'qualified_only'}
VAR_GLOBAL
	Sensor_Dis : ARRAY [0..10,0..100] OF UDINT;
	
	MovePos: ARRAY [0..50] OF LREAL := [500, 1000, 1500, 2000, 2500, 3000, 3500, 4000, 4500, 5000, 5500, 6000, 6500, 7000, 7500, 8000, -10, 34(0.0)];
	
	posCount	:INT;
	
	posCountMax: INT := 17;
	
	CycleCount : INT;
END_VAR

// ---- GVLs/AxisTest.TcGVL
{attribute 'qualified_only'}
VAR_GLOBAL
	test_Action_List : ARRAY [0..10] OF TestAction;
	
	pos :  ARRAY [0..3] OF LREAL;
END_VAR

// ---- GVLs/SpdC.TcGVL
{attribute 'qualified_only'}
VAR_GLOBAL PERSISTENT
// 上行架水平軸
	// 手動模式速度
	Jog_Speed :LREAL;
	// 手動模式加速度
	Jog_Accelerated :LREAL;
	// 手動模式減速度
	Jog_Deceleration :LREAL;
	
	// 自動模式 FX軸高速
	HighSpeed_FX :LREAL;
	// 自動模式高速
	HighSpeed :LREAL;
	// 自動模式低速
	LowSpeed :LREAL;
	// 回原點速度
	HomeSpeed :LREAL;
	// 離開原點速度
	DotSpeed :LREAL;
	// 手動模式加速度
	Accelerated :LREAL;
	// 手動模式減速度
	Deceleration :LREAL;

END_VAR

// ---- MSG/訊息列表/MsgBuff.TcGVL
{attribute 'qualified_only'}
VAR_GLOBAL
	// 儲列使用計數器
	evenNumber		: UDINT;
	
	DoneNumber 		: UDINT;

	messageList : ARRAY[0..15] OF MsgStruct;
	
// SQL 執行命令型
_fb_PLCDBCmdEvt : FB_PLCDBCmdEvt(sNetID:= '', tTimeout:= T#5S );

	systime         : FB_LocalSystemTime;
	currentTime     : DT;
END_VAR

// ---- POUs/硬體控制/測距感應器/I_DisSensor.TcIO
INTERFACE I_DisSensor

PROPERTY Distance : LREAL
GET
END_GET
END_PROPERTY

END_INTERFACE

// ---- POUs/硬體控制/軸/I_Axis.TcIO
INTERFACE I_Axis

METHOD AbsMove : BOOL
VAR_INPUT
	// 目標位置
	_Position : LREAL;
	// 移動速度
	_Velocity : LREAL := 0;
END_VAR
END_METHOD

PROPERTY Axis_States : ST_AxisStatus
GET
END_GET
END_PROPERTY

METHOD Homing : BOOL
VAR_INPUT
END_VAR
END_METHOD

PROPERTY Pos : LREAL
GET
END_GET
END_PROPERTY

METHOD PowerOff : BOOL
VAR_INPUT
END_VAR
END_METHOD

METHOD PowerOn : BOOL
VAR_INPUT
END_VAR
END_METHOD

METHOD RelMove : BOOL
VAR_INPUT
	// 目標距離
	_Position : LREAL;
	
	// 移動速度
	_Velocity : LREAL := 0;
END_VAR
END_METHOD

METHOD SetLimit : BOOL
VAR_INPUT
END_VAR
END_METHOD

PROPERTY State : Sub_Step
GET
END_GET
END_PROPERTY

METHOD Stop : BOOL
VAR_INPUT
	Dec : LREAL := 0;
END_VAR
END_METHOD

END_INTERFACE

// ---- POUs/MAIN.TcPOU
PROGRAM MAIN
VAR
	
	boot :BOOL := TRUE;

	tm : TIME;


END_VAR

IF boot THEN
	boot:=FALSE;
END_IF


MaBaseState();

GetEtherSta();

Sensor();

AutoMain();

GroupFx();

ExpConver();

AxisAction();

tm := TO_TIME(MaCfg.LaserPrinter_Timeout);
// SQL 專案資料讀寫功能
ReadSQLData();

LogFx();

MsgMain();

LightTower();

Button();

GetEtherSta();

ACTION init:

END_ACTION

END_PROGRAM

// ---- POUs/安全控制/MaBaseState.TcPOU
PROGRAM MaBaseState
VAR
//	msg: MsgPush;
	
	
	trig1: F_TRIG;
	trig2: F_TRIG;
	tmrEstop: TOF;
	ldp: R_TRIG;
	tmpState: MachineState;
	bDoorLock: BOOL;
	carDoor: BOOL;
	E_stop_trig1: F_TRIG;
	E_stop_trig2: F_TRIG;
	Door_trig1: F_TRIG;
	Door_trig2: F_TRIG;
	
	// 維修門切換延遲
	doorDelay: TOF;
	Door1_alarm_set: BOOL;
	Door2_alarm_set: BOOL;
	doorDelay1: TOF;
	tmr_Door_Car_Around: TOF;
	E_stop_trig3: F_TRIG;
	boot_tmr: TON := (IN := TRUE, PT := TIME#2s0ms);
END_VAR

IF boot_tmr.q THEN
	E_Stop();
	
	IF Estop THEN
		hmi.State := MachineState.emergency;
	ELSIF Door THEN
		hmi.State := MachineState.Door;
	ELSIF SystemError THEN
		hmi.State := MachineState.error;
	ELSIF NOT AutoMain.bBuzy THEN
		hmi.State := MachineState.standby;
	ELSIF AutoMain.bBuzy AND AutoMain.step >= 8000 AND AutoMain.step < 10000 THEN
		hmi.State := MachineState.manual_mode;
	END_IF
	
	IF hmi.SysErrorRest THEN
		SystemError :=FALSE;
		
		IF NOT SystemError THEN
			hmi.SysErrorRest := FALSE;
		END_IF
	END_IF
ELSE
	boot_tmr();
END_IF

ACTION E_Stop:
//	========================================
//					緊急停止				
//	========================================

Estop := NOT(IO.i101);

//// 緊急停止
E_stop_trig1(clk:=IO.i616); 
IF E_stop_trig1.Q THEN
	pMsg.Push_Error("緊急停止 MPG");
END_IF

E_stop_trig2(clk:=IO.i101); 
IF E_stop_trig2.Q AND NOT SystemError THEN
	pMsg.Push_Error("緊急停止 面板");
END_IF

//E_stop_trig2(clk:=io0.X002 AND io0.X003); 
//IF E_stop_trig2.Q THEN
//	pMsg.Push_Error("緊急停止 台車面板");
//END_IF

//E_stop_trig3(clk:=io0.X101); 
//IF E_stop_trig3.Q THEN
//	pMsg.Push_Error("緊急停止 台車");
//END_IF
END_ACTION

END_PROGRAM

// ---- POUs/動作流程控制/AutoMain.TcPOU
PROGRAM AutoMain
VAR
	
	step: DINT;
	
	// 自動執行中 的 進料動作流程
	step_Feed: Sub_Step;
	
	startStep: DINT;

	PutFloor: UINT;
	GetFloor: UINT;
	tmr01: TON;
	tmr8000: TON;
	Jog_Ldp: ARRAY[0..15] OF R_TRIG;

	fbWritePersistentData: FB_WritePersistentData;


	tmr_ErrorReset: TON;
	tmr_AutoLock: TON;
	
	sFilename: ARRAY [1..9] OF STRING := ['TEST-100-1', 'TEST-100-2', 'TEST-100-3', 'TEST-100-4', 'TEST-100-5', 'TEST-100-6', 'TEST-100-7', 'TEST-100-8', 'TEST-100-9'];
	fPoint: ARRAY [1..9, 1..2] OF REAL := [2(0.0), 100, 0.0, 100, 0.0, -200, 2(100), 0.0, 100, 0.0, -200, 2(100), 0.0, 100, 0.0];
	
	fPoint2: ARRAY [1..4, 1..2] OF REAL := [2(0.0), 80, 0.0, 80, 3(0)];
	
	fPointStart: ARRAY [1..2] OF REAL;
	
	iCount : INT;
	posCount: INT;
	
	NowWidth : LREAL;
	i: DINT;
	
	// 上次取得位置
	Last_Pos: LREAL;
	MaxWidth: LREAL;
	MinWidth: LREAL;
	FormatString: FB_FormatString2;
	
	_debug_X_NextPos_count :INT;
	_debug_X_NextPos : ARRAY [0..99] OF LREAL;
	
	// 軸組B雷射的距離
	GroupB_Now_Z: LREAL;
	// 回原點模式
	homeMode: BOOL;
	
	// A、C 能找到的 X保留位置
	LastXCanFind	:	LREAL;
	
	_log : Step_Log; 
	// SQL請求序號
	sql_hand: UDINT;
	
	
END_VAR

VAR_OUTPUT
	bBuzy: BOOL;
	bError: BOOL;
	bDone: BOOL;
	iErrorId : DINT;
END_VAR

WebHmi();

GroupA();
GroupB();
GroupC();
GroupD();

IF (EStop OR SystemError) AND bBuzy THEN
	hmi.Auto_bDone := FALSE;
	IF bBuzy THEN
		step := step  + 10000;
	END_IF
END_IF

bBuzy := (step >= 100 AND step < 10000);
bError := (step > 10000);

tmr_ErrorReset(in:= bError, PT:=T#1S);

IF tmr_ErrorReset.Q THEN
	iErrorId := step;
	step := 0;
END_IF




IF (ProgramReset OR Safety.SystemError) AND bError THEN
	step := 0;
END_IF

Step_0_Main();
step_0100_Homming();
step_0500_AutoMode_StartCheck();
step_0600_AutoMode_Feed();
step_0700_AutoMode_GoPrintPoint();
step_0800_AutoMode_GoPrintPoint_Cycle_200_UP();
step_0900_AutoMode_GoPrintPoint_Cycle_200_Down();
step_1000_AutoPrgEnd();

Start_Feed_In_NC_Start();

step_7800_FindZ();
step_8000_Jog();

TestActionPou();


// IF (bError) THEN
// 	hmi.Auto_Start := FALSE;
// 	hmi.Auto_Pause := FALSE;
// 	iErrorId := step - 10000;
// END_IF

Timer();
WritePersistentData();

_log(name := 'AutoMain', step := step);

METHOD Homming
VAR_INPUT
END_VAR
step := 100;
END_METHOD

METHOD JogMode
VAR_INPUT
END_VAR
step := 8000;
END_METHOD

METHOD JogMode_Exit
VAR_INPUT
END_VAR
step := 9800;
END_METHOD

METHOD ReStart
VAR_INPUT
END_VAR
step := 600;
END_METHOD

ACTION Start_Feed_In_NC_Start:

IF step > 700 AND step < 1000 AND	// 自動流程進入加工階段
	NOT step_Feed.bBuzy AND 		// 動作中進料沒在執行
	NOT ExpConver.Feed_bBuzy		// 進料機沒在執行
	THEN
		IF Hmi_Web.Auto_Start THEN
			step_Feed.Step := 1;
		END_IF
END_IF

CASE step_Feed.Step OF
	1:
		IF 	NOT ReadSQLData.bBuzy THEN
			step_Feed.Step := step_Feed.Step + 1;
		END_IF

	2:	// 從資料庫讀取是否有等待中的料
		sql_hand := ReadSQLData.Get_Steel_Num_On_Wait();
		IF sql_hand <> 0 THEN
			step_Feed.Step := step_Feed.Step + 1;
		END_IF
		
	3:
		IF ReadSQLData.bBuzy OR ReadSQLData.bError THEN
			step_Feed.Step := step_Feed.Step + 1;
		END_IF
			
	4:
		IF ReadSQLData.bDone = sql_hand THEN
			step_Feed.Step := step_Feed.Step + 1;
		ELSIF ReadSQLData.bError THEN
			step_Feed.Step := step_Feed.Step + 10000;
		END_IF
		
	5:
		IF ProjectData.WorkOrder_Num_On_Wait > 0 THEN
			// 有等待中的料
			step_Feed.Step := step_Feed.Step + 1;
		ELSE
			// 沒有等待中的料，關閉 Hmi_Web.Auto_Start 並 結束流程
			Hmi_Web.Auto_Start := FALSE;
			step_Feed.Step := 0;
		END_IF
		
	6:
		step_Feed.Step := 10;
		
	
	10: // 自動流程還在 加工中 的狀態
		IF step > 700 AND step < 1000 THEN
			// 啟動 自動進料機
			ExpConver.Feed_holding_2_waitLoading();
			// 關閉 Hmi_Web.Auto_Start 的訊號
			Hmi_Web.Auto_Start := FALSE;
			step_Feed.Step := step_Feed.Step + 1;
		ELSE
			// 加工已經結束
			step_Feed.Step := 0;
		END_IF
		
	11:
		IF ExpConver.Feed_bBuzy OR ExpConver.Feed_bError THEN
			step_Feed.Step := step_Feed.Step + 1;
		END_IF
		
	12:
		step_Feed.Step := 0;
		step_Feed.bDone := TRUE;
		
	
		
END_CASE

step_Feed.bBuzy := step_Feed.Step > 0 AND step_Feed.Step < 10000;
step_Feed.bError := step_Feed.Step > 10000;
IF step_Feed.bBuzy OR step_Feed.bError THEN
	step_Feed.bDone := FALSE;
END_IF
END_ACTION

ACTION Step_0_Main:
(*======================================
		確認起動條件&回原點
  ======================================*)
// 處裡緊急停止訊號
CASE step OF
	0:
		Button.StopButton_Light := 0;
		Button.StartButton_Light := 0;
		IF Hmi_Web.Jog_Mode THEN
			Hmi.Jog_Mode := FALSE;
			Hmi_Web.Jog_Mode := FALSE;
			SystemError := FALSE;
			IF NOT SystemError THEN
				step := 8000;
			END_IF
		ELSIF Hmi_Web.MPG_Mode THEN
			Hmi.MPG_Mode := FALSE;
			SystemError := FALSE;
			IF NOT SystemError THEN
				step := 8010;
			END_IF
		ELSIF Hmi_Web.Auto_Start OR Hmi_Web.Auto_OneCycle_Start THEN
// 			Hmi_Web.Auto_Start := FALSE;
// 			Hmi_Web.Auto_OneCycle_Start  := FALSE;
			IF NOT SystemError THEN
				step := 1;
			ELSE
				Hmi_Web.Auto_Start := FALSE;
				Hmi_Web.Auto_OneCycle_Start  := FALSE;
			END_IF
		END_IF
		
	
	1:
		// 檢查是否有設定要啟動的程式
		IF SystemError THEN
			Hmi_Web.Auto_Start := FALSE;
			Hmi_Web.Auto_OneCycle_Start := FALSE;
		ELSIF Hmi_Web.Auto_Start OR Hmi_Web.Auto_OneCycle_Start THEN
			step := step + 1;
		END_IF
		
	2:
		IF NOT GrobelVariable.bHome OR GbZ.fPos < 490 THEN
			step := 100;
		ELSE
			step := 500;
		END_IF
		
		

		
		
	10:
		
		tmr01.PT := T#500MS;
		tmr01.IN := TRUE;
		IF tmr01.Q THEN
			tmr01.IN := FALSE;
			step := step + 1;
		END_IF
		
	11:
		SystemError := FALSE;
		IF Hmi.Mode_Select = 1 THEN
			step := 8000;
		ELSIF Hmi.Mode_Select = 2 THEN
			step := 8010;
		ELSE
			step := 0;
		END_IF
		

// ============== 動作結束 ==============

	
	
	9900:
		hmi.Auto_bDone:=TRUE;
		hmi.Auto_Start := FALSE;
		hmi.Auto_ProgramSelect := 0;
		fbWritePersistentData.START := TRUE;
		step := step  + 1;
		
		
	9901:
		uRunCounter := uRunCounter + 1;
		step := step  + 1;
		
	9902:
		IF NOT fbWritePersistentData.BUSY THEN
			fbWritePersistentData.START := FALSE;
			step := step  + 1;
		END_IF
		
	9903:
		step := 0;
		
	9905:
		hmi.Auto_Start := false;
		hmi.Auto_ProgramSelect := 0;
		PutFloor := 0;
		GetFloor := 0;
		step := step  + 1;
		
	9906:
		
		step := 0;
		
	9910:
		GaX.PowerOff();
		GaY.PowerOff();
		GaZ.PowerOff();
		GbX.PowerOff();
		GbY.PowerOff();
		GbZ.PowerOff();
		GcX.PowerOff();
		GcY.PowerOff();
		GcZ.PowerOff();
		GdX.PowerOff();
		GdY.PowerOff();
		GdZ.PowerOff();
		step := 0;
		
END_CASE

IF step = 0 THEN
	RETURN;
END_IF

// step_7900_SensorTest();
END_ACTION

ACTION step_0100_Homming:
CASE step OF
	100:
		Button.HomeButton_Light := 2;
		step := 110;

	110:
		GroupA.ToStanby();
		GroupB.ToStanby();
		GroupC.ToStanby();
		GroupD.ToStanby();
		step := step + 1;
		
	111:
		IF (GroupA.StepA.bBuzy OR GroupA.StepA.bError) AND 
			(GroupB.StepA.bBuzy OR GroupB.StepA.bError) AND
			(GroupC.StepA.bBuzy OR GroupC.StepA.bError) AND
			(GroupD.StepA.bBuzy OR GroupD.StepA.bError) THEN
				step := step + 1;
		END_IF
		
	112:
		IF ExpConver.Feed_bBuzy THEN
			ExpConver.Feed_Reset();
		ELSE
			step := 114;
		END_IF
		
	113:
		IF NOT ExpConver.Feed_bBuzy AND NOT ExpConver.ExpConver_Reset THEN
			step := step + 1;
		END_IF
		
	114:
		ExpConver.FeedHomeStart();
		IF (ExpConver.Feed_bBuzy OR ExpConver.Feed_bError) THEN
			step := step + 1;
		END_IF

	115:
		IF GroupB.StepA.bDone THEN
			step := step + 1;
		ELSIF GroupA.StepA.bError OR GroupB.StepA.bError OR GroupC.StepA.bError OR GroupD.StepA.bError THEN
			step := step + 10000;
		END_IF
		
	116:
		step := 120;
		
		
	120:
		homeMode := (IO.i501 OR IO.i502 OR IO.i503 OR IO.i504) AND GroupFx.b_AC_HOME AND GroupFx.b_BD_HOME; 
		GroupFx.A_UnPress();
		GroupFx.B_UnPress();
		GroupFx.C_UnPress();
		GroupFx.D_UnPress();
		step := step + 1;
		
	121:
		IF (GroupFx.step_A_P.bBuzy OR GroupFx.step_A_P.bError) AND 
			(GroupFx.step_B_P.bBuzy OR GroupFx.step_B_P.bError) AND
			(GroupFx.step_C_P.bBuzy OR GroupFx.step_C_P.bError) AND
			(GroupFx.step_D_P.bBuzy OR GroupFx.step_D_P.bError) THEN
				step := step + 1;
		END_IF
		
	122:
		
		IF GroupFx.step_A_P.bDone AND GroupFx.step_B_P.bDone AND GroupFx.step_C_P.bDone AND GroupFx.step_D_P.bDone THEN
			step := step + 1;
		ELSIF GroupFx.step_A_P.bError OR GroupFx.step_B_P.bError OR GroupFx.step_C_P.bError OR GroupFx.step_D_P.bError THEN
			step := step + 10000;
		END_IF
		
	123:
		step := 130;
		
		
	130:
		IF homeMode THEN
			GroupFx.AC_UnClamp(10);
			GroupFx.BD_UnClamp(10);
		ELSE
			GroupFx.AC_Home();
			GroupFx.BD_Home();
		END_IF
		step := step + 1;
		
	131:
		IF (GroupFx.step_AC_C.bBuzy OR GroupFx.step_AC_C.bError) AND 
			(GroupFx.step_BD_C.bBuzy OR GroupFx.step_BD_C.bError) THEN
				step := step + 1;
		END_IF
		
	132:
		
		IF GroupFx.step_AC_C.bDone AND GroupFx.step_BD_C.bDone THEN
			step := step + 1;
		ELSIF GroupFx.step_AC_C.bError OR GroupFx.step_BD_C.bError THEN
			step := step + 10000;
		END_IF
		
	133:
		step := 140;
		
	140:
		IF NOT GroupFx.b_AC_HOME THEN
			GroupFx.AC_Home();
		END_IF
		IF NOT GroupFx.b_BD_HOME THEN
			GroupFx.BD_Home();
		END_IF
		step := step + 1;
		
	141:
		IF (GroupFx.step_AC_C.bBuzy OR GroupFx.step_AC_C.bError OR GroupFx.b_AC_HOME) AND 
			(GroupFx.step_BD_C.bBuzy OR GroupFx.step_BD_C.bError OR GroupFx.b_BD_HOME) THEN
				step := step + 1;
		END_IF
		
	142:
		IF (GroupFx.step_AC_C.bDone OR GroupFx.b_AC_HOME) AND (GroupFx.step_BD_C.bDone OR GroupFx.b_BD_HOME) THEN
			step := step + 1;
		ELSIF GroupFx.step_AC_C.bError OR GroupFx.step_BD_C.bError THEN
			step := step + 10000;
		END_IF	
		
	143:
		step := 150;
		
	150:
		IF ExpConver.Feed_bDone THEN
			step := step + 1;
		ELSIF ExpConver.Feed_bError THEN
			step := step + 10000;
			pMsg.Push_Error("自動料架復歸時發生錯誤");
		END_IF
		
	151:
		IF GroupA.StepA.bDone AND GroupC.StepA.bDone AND GroupC.StepA.bDone THEN
			step := step + 1;
		ELSIF GroupA.StepA.bError AND GroupC.StepA.bError AND GroupC.StepA.bError THEN
			step := step + 10000;
			pMsg.Push_Error("自動料架復歸時發生錯誤");
		END_IF
		
	152:
		Button.HomeButton_Light := 1;
		bDone := TRUE;
		GrobelVariable.bHome := TRUE;
		step := 0;
END_CASE
END_ACTION

ACTION step_0500_AutoMode_StartCheck:
CASE step OF
(*	====================================
				啟動前檢查
	====================================*)
		500:
			hmi.State := MachineState.auto_mode;
			IF IO.i212 THEN
				step := step + 1;
			ELSE
				pMsg.Push_Alarm_NoPause("氣壓壓力不足");
				step := 0;
			END_IF
			
		501:
			step := 510;
			
			
(*	================================================
			讀取 資料庫 的 work_order 資料表
	================================================*)
		510:
			sql_hand := ReadSQLData.Get_WorkkOrder();
			IF sql_hand <> 0 THEN
				step := step + 1;
			END_IF
			
		511:
			IF ReadSQLData.bBuzy OR ReadSQLData.bError THEN
				step := step + 1;
			END_IF
			
		512:
			IF ReadSQLData.bDone = sql_hand THEN
				step := step + 1;
			ELSIF ReadSQLData.bError THEN
				step := step + 10000;
			END_IF
			
		513:
			IF Hmi_Web.Auto_Start THEN 
				
				// 標準進料模式
				Hmi_Web.Auto_Start := FALSE;
				step := 520;
			ELSIF Hmi_Web.Auto_OneCycle_Start THEN
				
				// 插單模式
				Hmi_Web.Auto_OneCycle_Start := FALSE;
				step := step + 1;
			END_IF
			
		514: // 插單模式 檢查 插單 或 不靠邊插單 是否有資料
			IF LEN(STR:=ProjectData.WorkOrder_inserts.steel_id) > 0 OR
				LEN(STR:=ProjectData.WorkOrder_alignment.steel_id) > 0
			THEN
				
				step := 550;
			ELSE
				pMsg.Push_Error(
					WStrConcat(
					str0:= "找不到 插單 或 不靠邊插單 的資料 AutoMain:", 
					str1:= TO_WSTRING(step))
				);
			END_IF
				
				
(*	====================================
				標準進料模式
	====================================*)
		520:
			IF LEN(STR:=ProjectData.WorkOrder_inSide.steel_id) > 0 THEN
				// 已經有 料的狀態 是 在輸送滾輪上(inSide)
				ProjectData.WorkOrder_Now := ProjectData.WorkOrder_inSide;
				step := step + 1;
			ELSE
				// 沒有 料的狀態 是 在輸送滾輪上(inSide)
				step := 530;
			END_IF
			
		521: // 自動進料機執行搬移動作，但不進料到 輸送滾輪上
			ExpConver.Feed_holding_2_waitLoading();
			step := step + 1;
			
		522:
			IF ExpConver.Feed_bBuzy OR ExpConver.Feed_bError THEN
				step := step + 1;
			END_IF
			
		523: // 確認自動進料機執行後，繼續機器進料動作
			step := 570;
			
(*	========================================
		標準進料模式 - 沒有料在輸送滾輪上
	========================================*)
		530: // 自動進料機 執行完整進料
			ExpConver.FeedAutoStart();
			step := step + 1;
			
		531:
			IF ExpConver.Feed_bBuzy OR ExpConver.Feed_bError THEN
				step := step + 1;
			END_IF
			
		532:
			IF ExpConver.Feed_bDone THEN
				step := step + 1;
			ELSIF ExpConver.Feed_bError THEN
				step := step + 10000;
			END_IF
			
		533:
			step := 540;
			
(*	========================================
		進料結束後 再次讀取資料庫
	========================================*)
		540:
			sql_hand := ReadSQLData.Get_WorkkOrder();
			IF sql_hand <> 0 THEN
				step := step + 1;
			END_IF
			
		541:
			IF ReadSQLData.bBuzy OR ReadSQLData.bError THEN
				step := step + 1;
			END_IF
			
		542:
			IF ReadSQLData.bDone = sql_hand THEN
				step := step + 1;
			ELSIF ReadSQLData.bError THEN
				step := step + 10000;
			END_IF
			
		543:
			IF LEN(STR:=ProjectData.WorkOrder_inSide.steel_id) > 0 THEN
				// 已經有 料的狀態 是 在輸送滾輪上(inSide)
				ProjectData.WorkOrder_Now := ProjectData.WorkOrder_inSide;
				step := step + 1;
			ELSE
				// 沒有 料的狀態 是 在輸送滾輪上(inSide)
				pMsg.Push_Error(
					WStrConcat(
					str0:= "找不到狀態是 輸送滾輪上(inSide) 的資料 AutoMain:", 
					str1:= TO_WSTRING(step))
				);
			END_IF
			
		544:
			step := 570;
			
(*	=======================================
				插單模式 
			料已放置在 輸送滾輪 上
	=======================================*)
		550:
			sql_hand := ReadSQLData.Get_WorkkOrder();
			IF sql_hand <> 0 THEN
				step := step + 1;
			END_IF
			
		551:
			IF (ReadSQLData.bBuzy OR ReadSQLData.bError) THEN
				step := step + 1;
			END_IF
			
		552:
			IF ReadSQLData.bDone = sql_hand THEN
				step := step + 1;
			ELSIF ReadSQLData.bError THEN
				step := step + 10000;
			END_IF
			
		553:
			step := 560;
			
			
		560:
			IF LEN(STR:=ProjectData.WorkOrder_alignment.steel_id) > 0 THEN
				// 無靠邊差單
				ProjectData.WorkOrder_Now := ProjectData.WorkOrder_alignment;
				step := step + 1;
			ELSIF LEN(STR:=ProjectData.WorkOrder_inserts.steel_id) > 0 THEN
				// 差單
				ProjectData.WorkOrder_Now := ProjectData.WorkOrder_inserts;
				step := step + 1;
			ELSE
				pMsg.Push_Error("AutoMain: 無差單資料");
				step := 0;
			END_IF
			
			
		561:
			step := 570;

(*	=======================================
			從資料庫 讀取 材料資料
	=======================================*)
		570:
			sql_hand := ReadSQLData.Get_SteelData(ProjectData.WorkOrder_Now.steel_id);
			IF sql_hand <> 0 THEN
				step := step + 1;
			END_IF
			
		571:
			IF ReadSQLData.bBuzy OR ReadSQLData.bError THEN
				step := step + 1;
			END_IF
			
		572:
			IF ReadSQLData.bDone = sql_hand THEN
				step := step + 1;
			ELSIF ReadSQLData.bError THEN
				step := step + 10000;
			END_IF
			
		573:
			IF LEN(STR:=ProjectData.WorkOrder_alignment.steel_id) > 0 THEN
				// 無靠邊差單
				step := 590;
			ELSIF LEN(STR:=ProjectData.WorkOrder_inserts.steel_id) > 0 THEN
				// 差單
				step := 580;
			ELSIF LEN(STR:=ProjectData.WorkOrder_inSide.steel_id) > 0 THEN
				// 料架進料
				step := 600;
			END_IF
			
			
(*	=======================================
			等待按下 機器啟動
	=======================================*)		
		580:
			hmi.State := MachineState.auto_mode_wait;
			Button.StartButton_Light := 2;
			step := step + 1;
			
		581:
			
			IF Button.StartButton THEN
				step := step + 1;
			END_IF
			
		582:
			hmi.State := MachineState.auto_mode;
			Button.StartButton_Light := 1;
			step := 590;		

	
(*	=======================================
					靠邊
	=======================================*)	
		590:
			ExpConver.Feed_PullOver();
			step := step + 1;
			
		591:
			IF ExpConver.Feed_bBuzy OR ExpConver.Feed_bError THEN
				step := step + 1;
			END_IF
			
		592:
			IF ExpConver.Feed_bDone THEN
				step := step + 1;
			ELSIF ExpConver.Feed_bError THEN
				step := step + 10000;
			END_IF
			
		593:
			step := 600;
			
		

			
END_CASE
END_ACTION

ACTION step_0600_AutoMode_Feed:
CASE step OF
(*	==================================================
			夾輪到指定位置（防止工件墬落）
	==================================================*) 
	600: 
		ExpConver.InRollerStop();
		NowWidth := ProjectData.Now_Steel.Height;
		step := step + 1;
		
	601:
		// 側夾開到 工件寬度 + 15 的位置
		GroupFx.AC_Clamp(NowWidth + 15);
		GroupFx.BD_Clamp(NowWidth + 15);
		// 下壓動作確認 工件高度 > 上次工件高度 + 5，升起下壓
		IF ProjectData.Now_Steel.Width > ProjectData.old_Steel.Width + 5 THEN
			GroupFx.A_UnPress();
			GroupFx.B_UnPress();
			GroupFx.C_UnPress();
			GroupFx.D_UnPress();
		END_IF
		step := step + 1;
		
	602:
		IF (GroupFx.step_AC_C.bBuzy OR GroupFx.step_AC_C.bError) AND
			(GroupFx.step_BD_C.bBuzy OR GroupFx.step_BD_C.bError) THEN
			step := step + 1;
		END_IF
		
	603:
		step := 610;
(*	==================================================
			材料進入 入口位置 測量寬度
	==================================================*) 
	610:// 材料進入 入口位置
		ExpConver.InRollerStart();
		step := step + 1;
		
	611:
		IF ExpConver.In_Moter_Running OR ExpConver.In_Moter_Error THEN
			step := step + 1;
		END_IF
		
	612: // 到達 入口感應器 後停止
		IF io.i711 OR ExpConver.In_Moter_Error THEN
			// 停止馬達
			ExpConver.InRollerStop();
			
			IF  io.i711 THEN
				step := step + 1;
			ELSIF ExpConver.In_Moter_Error THEN
				pmsg.Push_Error(
					WStrConcat("AutoMain:進料馬達發生錯誤", TO_WSTRING(step))
				);
				step := step + 10000;
			END_IF
		END_IF
		
	613: // 確認進料馬達停止
		tmr01.PT := T#2S;
		tmr01.IN := NOT ExpConver.In_Moter_Running;
		IF tmr01.Q THEN
			tmr01.IN := FALSE;
			step := step + 1;
		END_IF
		
	614:// 紀錄寬度數據
	
		MaxWidth := ProjectData.Now_Steel.Height + (ProjectData.Now_Steel.Height * 0.2); 
		MinWidth := ProjectData.Now_Steel.Height - (ProjectData.Now_Steel.Height * 0.2);
		IF ExpConver.Feed_Workpiace_H > MinWidth AND ExpConver.Feed_Workpiace_H < MaxWidth THEN
			step := step + 1;
		ELSE
			pMsg.Push_Error(WStrConcat(
				"AutoMain: ",
				WLEFT(STR:= TO_WSTRING(ProjectData.Now_Steel.uid), SIZE:= 8),
				" :高度數據與輸入資料錯誤,設定值:",
				TO_WSTRING(NowWidth),
				" 實際值:",
				TO_WSTRING(ExpConver.Feed_Workpiace_H)
				));
			step := step + 10000;
		END_IF
// 		HightCheck(ExpConver.Feed_Workpiace_H, ExpConver.Feed_Workpiace_W);
		
		
	615:
		IF GroupFx.step_AC_C.bDone AND GroupFx.step_BD_C.bDone THEN
			step := step + 1;
		ELSIF GroupFx.step_AC_C.bError OR GroupFx.step_BD_C.bError THEN
			step := step + 10000;
		END_IF
		
	616:
		step := 630;
(*	==================================================
			材料前進到 出口位置 (整料)
	==================================================*) 
	630:
		ExpConver.InRollerStart();
		step := step + 1;
		
	631:
		IF ExpConver.In_Moter_Running OR ExpConver.In_Moter_Error THEN
			step := step + 1;
		END_IF
		
	632: // 到達 出口感應器 後停止
		IF io.i709 OR ExpConver.In_Moter_Error THEN
			// 停止馬達
			ExpConver.InRollerStop();
			
			IF  io.i709 THEN
				step := step + 1;
			ELSIF ExpConver.In_Moter_Error THEN
				pmsg.Push_Error(
					WStrConcat("AutoMain:進料馬達發生錯誤", TO_WSTRING(step))
				);
				step := step + 10000;
			END_IF
		END_IF
		
	633: // 確認進料馬達停止
		tmr01.PT := T#2S;
		tmr01.IN := NOT ExpConver.In_Moter_Running;
		IF tmr01.Q THEN
			tmr01.IN := FALSE;
			step := step + 1;
		END_IF
		
	634:
		step := 640;
		
		
(*	=========================
			整料開始
	=========================*) 
	640: // BD
		GroupFx.AC_Clamp(0);
		GroupFx.BD_Clamp(0);
		step := step + 1;
	
	641:
		IF (GroupFx.step_AC_C.bBuzy OR GroupFx.step_AC_C.bError) AND
			(GroupFx.step_BD_C.bBuzy OR GroupFx.step_BD_C.bError) THEN
			step := step + 1;
		END_IF
		
		
	642:
		IF GroupFx.step_AC_C.bDone AND GroupFx.step_BD_C.bDone THEN
			step := step + 1;
		ELSIF GroupFx.step_AC_C.bError OR GroupFx.step_BD_C.bError THEN
			step := step + 10000;
		END_IF
		
	643:
		step := 650;
		
		

	650:
		GroupFx.B_Press();
		GroupFx.D_Press();
		step := step + 1;
	
	651:
		IF (GroupFx.step_B_P.bBuzy OR GroupFx.step_B_P.bError) AND
			(GroupFx.step_D_P.bBuzy OR GroupFx.step_D_P.bError)
			THEN
			step := step + 1;
		END_IF
		
		
	652:
		IF GroupFx.step_B_P.bDone AND GroupFx.step_D_P.bDone THEN
			step := step + 1;
		ELSIF GroupFx.step_B_P.bError OR GroupFx.step_D_P.bError THEN
			step := step + 10000;
		END_IF
		
	653:
		step := 670;

(*	===============================================
			整料結束，退開 AC下壓 與 AC夾輪
	===============================================*) 
	660:
		GroupFx.A_UnPress();
		GroupFx.C_UnPress();
		step := step + 1;
	
	661:
		IF (GroupFx.step_A_P.bBuzy OR GroupFx.step_A_P.bError) AND
			(GroupFx.step_C_P.bBuzy OR GroupFx.step_C_P.bError) THEN
			step := step + 1;
		END_IF
		
		
	662:
		IF GroupFx.step_A_P.bDone AND GroupFx.step_C_P.bDone THEN
			step := step + 1;
		ELSIF GroupFx.step_A_P.bError OR GroupFx.step_C_P.bError THEN
			step := step + 10000;
		END_IF
		
	663:
		step := 670;
		
	670: // 退開 AC夾輪
		GroupFx.AC_UnClamp(10);
		step := step + 1;
	
	671:
		IF (GroupFx.step_AC_C.bBuzy OR GroupFx.step_AC_C.bError) THEN
			step := step + 1;
		END_IF
		
		
	672:
		IF GroupFx.step_AC_C.bDone THEN
			step := step + 1;
		ELSIF GroupFx.step_AC_C.bError THEN
			step := step + 10000;
		END_IF
		
	673:
		step := 680;


(*	============================
			工件原點整定
	============================*) 
	680:
		GroupFx.Fx_Home();
		step := step + 1;
		
	681:
		IF (GroupFx.bBuzy OR GroupFx.bError) THEN
			step := step + 1;
		END_IF
		
		
	682:
		IF GroupFx.bDone THEN
			step := step + 1;
		ELSIF GroupFx.bError THEN
			step := step + 10000;
		END_IF
	
	683:
		step := 690;
		
(*	============================
		工件進料結束 標示進料結束
	============================*) 
	690:
		Last_Pos := 0;
		sql_hand := ReadSQLData.Set_Steel_Start(ProjectData.Now_Steel.uid);
		IF sql_hand <> 0 THEN
			step := step + 1;
		END_IF
		
	691:
		IF ReadSQLData.bBuzy OR ReadSQLData.bError THEN
			step := step + 1;
		END_IF
			
	692:
		IF ReadSQLData.bDone = sql_hand THEN
			step := step + 1;
		ELSIF ReadSQLData.bError THEN
			step := step + 10000;
		END_IF
		
	693:
		step := 700;
END_CASE
END_ACTION

ACTION step_0700_AutoMode_GoPrintPoint:
CASE step OF
(*	===================================
				搜尋 X工作點
	===================================*)
	700:
		sql_hand := ReadSQLData.Get_X_NextPos(0);
		IF sql_hand <> 0 THEN
			step := step + 1;
		END_IF
		
	701:
		IF ReadSQLData.bBuzy OR ReadSQLData.bError THEN
			step := step + 1;
		END_IF
		
	702:
		IF ReadSQLData.bDone = sql_hand THEN
			step := step + 1;
		ELSIF ReadSQLData.bError THEN
			step := step + 10000;
		END_IF
		
	703:
		Last_Pos := ReadSQLData.fNext_XPos;
		// ============ 紀錄啟動條件 ============
		_log.fbJson.StartObject();
		_log.fbJson.AddKeyString('StepName','Get_Next_XPos');
		_log.fbJson.AddKeyLreal('fNext_XPos', Last_Pos);
		_log.JsonOutput();
		// ======================================
		_debug_X_NextPos[_debug_X_NextPos_count] := Last_Pos;
		_debug_X_NextPos_count := 1;
		step := step + 1;
		
	704:
		step := 710;
		
(*	==========================================
				取得區間的打標工作
	==========================================*)
	710:
		IF ProjectData.Now_Steel.Height > 200 THEN
			sql_hand := ReadSQLData.Get_Payload(Start_Pos := Last_Pos, End_Pos := Last_Pos + 200);
		ELSE
			sql_hand := ReadSQLData.Get_Payload(Start_Pos := Last_Pos, End_Pos := Last_Pos + 75);
		END_IF
		IF sql_hand <> 0 THEN
			step := step + 1;
		END_IF
		
	711:
		IF ReadSQLData.bBuzy OR ReadSQLData.bError THEN
			step := step + 1;
		END_IF
		
	712:
		IF ReadSQLData.bDone = sql_hand THEN
			step := step + 1;
		ELSIF ReadSQLData.bError THEN
			step := step + 10000;
		END_IF
		
	713:
		step := 720;

(*	==========================================
			設定各軸組 並 預移到打標點
	==========================================*)
	720: // 設定 各軸組 X參考座標
		GroupA.Set_X_Ref(Value := Last_Pos);
		GroupB.Set_X_Ref(Value := Last_Pos);
		GroupC.Set_X_Ref(Value := Last_Pos);
		GroupD.Set_X_Ref(Value := Last_Pos);
		step := step + 1;
		
	721: // 設定 各軸組 X參考座標
		GroupA.Set_Y_Ref(Value := MaCfg.laserA_Y_ReferencePos - ProjectData.Now_Steel.Width);
		GroupB.Set_Y_Ref(Value := MaCfg.laserB_Y_ReferencePos - ProjectData.Now_Steel.Height);
		GroupC.Set_Y_Ref(Value := MaCfg.laserC_Y_ReferencePos);
		GroupD.Set_Y_Ref(Value := MaCfg.laserD_Y_ReferencePos);
		step := step + 1;
	
	722: // 關閉打標 (讓 流程暫停 在 開始打標 前)
		GroupA.ReadyToPrint := FALSE;
		GroupB.ReadyToPrint := FALSE;
		GroupC.ReadyToPrint := FALSE;
		GroupD.ReadyToPrint := FALSE;
		
		GroupA.ReadyToMove := FALSE;
		GroupB.ReadyToMove := FALSE;
		GroupC.ReadyToMove := FALSE;
		GroupD.ReadyToMove := FALSE;
		step := step + 1;
		

	
	723: // 載入區域工作內容 + 預移動開始
		GroupA.Do_WorkList();
		GroupB.Do_WorkList();
		GroupC.Do_WorkList();
		GroupD.Do_WorkList();
		step := step + 1;
		
	724:
		IF (GroupA.bBuzy OR GroupA.bError OR ProjectData.Now_Steel_Payload_A_DataNumber = 0) AND
			(GroupB.bBuzy OR GroupB.bError OR ProjectData.Now_Steel_Payload_B_DataNumber = 0) AND
			(GroupC.bBuzy OR GroupC.bError OR ProjectData.Now_Steel_Payload_C_DataNumber = 0) AND
			(GroupD.bBuzy OR GroupD.bError OR ProjectData.Now_Steel_Payload_D_DataNumber = 0) THEN
				step := step + 1;
		END_IF
		
	725:
		step := 730;
		
(*	================================
		出料輸送滾輪有工件未吊離
	================================*)
	730:
		IF ExpConver.Out_sensor > 1 AND Last_Pos > 500 THEN
			hmi.State := MachineState.auto_mode_wait;
			step := step + 1;
		ELSE
			step := 732;
		END_IF
		
	731:
		IF ExpConver.Out_sensor > 1 THEN
			Button.StartButton_Light := 0;
		ELSE
			Button.StartButton_Light := 2;
			IF Button.StartButton THEN
				step := step + 1;
			END_IF
		END_IF
		
		
	732:
		hmi.State := MachineState.auto_mode;
		Button.StartButton_Light := 1;
		step := 740;

(*	===================================
				Fx 前往 X工作點
	===================================*)
	740:
		GroupFx.Fx_Move(Last_Pos);
		GaZ.AbsMove(posc.GaZ_P_Limite, spdc.HighSpeed);
		step := step + 1;
		
	741:
		IF (GroupFx.bBuzy OR GroupFx.bError) AND (GaZ.bBuzy OR GaZ.bError) THEN
			step := step + 1;
		END_IF
		
		
	742:
		IF GroupFx.bDone AND GaZ.bDone THEN
			step := step + 1;
		ELSIF GroupFx.bError OR GaZ.bError THEN
			step := step + 10000;
		END_IF
		
	743:
		step := 750;
		
	750:
		
		GroupB.FindZ();
		GroupC.FindZ();
		GroupD.FindZ();
		step := step + 1;
		
	751:
		IF 	(GroupB.StepA.bBuzy OR GroupB.StepA.bError) AND
			(GroupC.StepA.bBuzy OR GroupC.StepA.bError) AND
			(GroupD.StepA.bBuzy OR GroupD.StepA.bError) THEN
				step := step + 1;
		END_IF
		
	752:
		IF 	(GroupB.StepA.bDone) AND
			(GroupC.StepA.bDone) AND 
			(GroupD.StepA.bDone) THEN
				GroupB_Now_Z := GroupB.Az.Pos;	// 記錄軸組B的雷射距離，小於200的料使用
			 	step := step + 1;
		ELSIF 
			(GroupB.StepA.bError) OR 
			(GroupC.StepA.bError) OR 
			(GroupD.StepA.bError) THEN
				step := step + 10000;
		END_IF
		
	753:
		GroupA.FindZ();
		
		step := step + 1;
		
	754:
		IF 	(GroupA.StepA.bBuzy OR GroupA.StepA.bError) THEN
				step := step + 1;
		END_IF
		
	755:
		IF 	(GroupA.StepA.bDone) THEN
			step := step + 1;
		ELSIF 
			(GroupA.StepA.bError) THEN
				step := step + 10000;
		END_IF
		
	756:
		GroupA.ReadyToMove := TRUE;
		GroupB.ReadyToMove := TRUE;
		GroupC.ReadyToMove := TRUE;
		GroupD.ReadyToMove := true;
		step := 760;
		
(*	=============================================
				開始各組區域打標
	=============================================*)
	760: 
		tmr01.PT := T#2S;
		tmr01.IN := NOT ExpConver.In_Moter_Running;
		IF tmr01.Q THEN
			tmr01.IN := FALSE;
			step := step + 1;
		END_IF
		
	761:
		GroupA.ReadyToPrint := TRUE;
		GroupB.ReadyToPrint := TRUE;
		GroupC.ReadyToPrint := TRUE;
		GroupD.ReadyToPrint := TRUE;
		step := step + 1;
		
	762:
		IF GroupA.bDone AND GroupB.bDone AND GroupC.bDone AND GroupD.bDone THEN
			step := step + 1;
		ELSIF GroupA.bError OR GroupB.bError OR GroupC.bError OR GroupD.bError THEN
			step := step + 10000;
		END_IF
		
	763:
		step := 770;
		
(*	================================
		出料輸送滾輪有工件未吊離
	================================*)
	770:
		IF ExpConver.Out_sensor > 1 AND Last_Pos < 500 THEN
			hmi.State := MachineState.auto_mode_wait;
			step := step + 1;
		ELSE
			step := 772;
		END_IF
		
	771:
		IF ExpConver.Out_sensor > 1 THEN
			Button.StartButton_Light := 0;
			Button.StopButton_Light := 2;
		ELSE
			Button.StartButton_Light := 2;
			Button.StopButton_Light := 0;
			IF Button.StartButton THEN
				step := step + 1;
			END_IF
		END_IF
		
		
	772:
		
		hmi.State := MachineState.auto_mode;
		Button.StartButton_Light := 1;
		IF ProjectData.Now_Steel.Height > 200 THEN
			step := 800;
		ELSE
			step := 900;
		END_IF
		
END_CASE
END_ACTION

ACTION step_0800_AutoMode_GoPrintPoint_Cycle_200_UP:
(*=====================================
				搜尋 X工作點
=======================================*)

CASE step OF
(*	===================================
				搜尋 X工作點
	===================================*)
	800:
		sql_hand := ReadSQLData.Get_X_NextPos(Last_Pos + 200);
		IF sql_hand <> 0 THEN
			step := step + 1;
		END_IF
		
	801:
		IF ReadSQLData.bBuzy OR ReadSQLData.bError THEN
			step := step + 1;
		END_IF
		
	802:
		IF ReadSQLData.bDone = sql_hand THEN
			step := step + 1;
		ELSIF ReadSQLData.bError THEN
			step := step + 10000;
		END_IF
		
	803:
		Last_Pos := ReadSQLData.fNext_XPos;
		
		// ============ 紀錄啟動條件 ============
		_log.fbJson.StartObject();
		_log.fbJson.AddKeyString('StepName','Get_Next_XPos');
		_log.fbJson.AddKeyLreal('fNext_XPos', Last_Pos);
		_log.JsonOutput();
		// ======================================
		
		_debug_X_NextPos[_debug_X_NextPos_count] := Last_Pos;
		_debug_X_NextPos_count := _debug_X_NextPos_count + 1;
		
		step := step + 1;
		
	804:
		IF Last_Pos = -1 THEN
			step := 1000;
		ELSE
			step := step + 1;
		END_IF
		
	805:
		step := 810;
		
(*	==========================================
				取得區間的打標工作
	==========================================*)
	810:
		sql_hand := ReadSQLData.Get_Payload(Start_Pos := Last_Pos, End_Pos := Last_Pos + 200);
		IF sql_hand <> 0 THEN
			step := step + 1;
		END_IF
		
	811:
		IF ReadSQLData.bBuzy OR ReadSQLData.bError THEN
			step := step + 1;
		END_IF
		
	812:
		IF ReadSQLData.bDone = sql_hand THEN
			step := step + 1;
		ELSIF ReadSQLData.bError THEN
			step := step + 10000;
		END_IF
		
	813:
		Last_Pos := Last_Pos - 10;
		step := 820;

(*	==========================================
			設定各軸組 並 預移到打標點
	==========================================*)
	820: // 設定 各軸組 X參考座標
		GroupA.Set_X_Ref(Value := Last_Pos);
		GroupB.Set_X_Ref(Value := Last_Pos);
		GroupC.Set_X_Ref(Value := Last_Pos);
		GroupD.Set_X_Ref(Value := Last_Pos);
		step := step + 1;
		
	821:
		GroupA.ReadyToPrint := FALSE;
		GroupB.ReadyToPrint := FALSE;
		GroupC.ReadyToPrint := FALSE;
		GroupD.ReadyToPrint := FALSE;
		
		GroupA.ReadyToMove := FALSE;
		GroupB.ReadyToMove := FALSE;
		GroupC.ReadyToMove := FALSE;
		GroupD.ReadyToMove := FALSE;
		step := step + 1;
		

	
	822: // 載入區域工作內容 + 預移動開始
		GroupA.Do_WorkList();
		GroupB.Do_WorkList();
		GroupC.Do_WorkList();
		GroupD.Do_WorkList();
		step := step + 1;
		
	823:
		IF (GroupA.bBuzy OR GroupA.bError OR ProjectData.Now_Steel_Payload_A_DataNumber = 0) AND
			(GroupB.bBuzy OR GroupB.bError OR ProjectData.Now_Steel_Payload_B_DataNumber = 0) AND
			(GroupC.bBuzy OR GroupC.bError OR ProjectData.Now_Steel_Payload_C_DataNumber = 0) AND
			(GroupD.bBuzy OR GroupD.bError OR ProjectData.Now_Steel_Payload_D_DataNumber = 0) THEN
				step := step + 1;
		END_IF
		
	824:
		step := 830;
		
(*	===================================
			判斷是否走快到結尾
			如果是則交換編碼器
	===================================*)
	830: // 判斷是否走快到結尾
		LastXCanFind := 10 + 75 + MAX(ABS(MaCfg.laserA_X_DisSensor2LaserCenter), ABS(MaCfg.laserC_X_DisSensor2LaserCenter)); // 計算 測高感應器 能照到的 X位置
		IF (Last_Pos + 1200) > ProjectData.Now_Steel.Length AND GroupFx.b_BD_Clamp THEN
			IF Fx.fPos < 1200 THEN
				step := step + 1;
			ELSE
				step := 835;
			END_IF
		ELSIF (Last_Pos + LastXCanFind) >= ProjectData.Now_Steel.Length THEN
			Last_Pos := Last_Pos - LastXCanFind;
			GroupA.Set_X_Ref(Value := Last_Pos);
			GroupB.Set_X_Ref(Value := Last_Pos);
			GroupC.Set_X_Ref(Value := Last_Pos);
			GroupD.Set_X_Ref(Value := Last_Pos);
			step := 850;
		ELSE
			step := 850;
		END_IF
		
		
	831:
		SensorTest.MovePos[0] := Sensor.sensor_test_pos;
		SensorTest.MovePos[1] := FxA_Exp_Pos;
		SensorTest.MovePos[2] := FxB_Exp_Pos;
		
		GroupFx.Fx_Move(1200);
		step := step + 1;
		
	832:
		IF (GroupFx.bBuzy OR GroupFx.bError) THEN
			step := step + 1;
		END_IF
		
		
	833:
		IF GroupFx.bDone THEN
			step := step + 1;
		ELSIF GroupFx.bError THEN
			step := step + 10000;
		END_IF
		
	834:
		step := 835;
		
	835:
		SensorTest.MovePos[4] := Sensor.sensor_test_pos;
		SensorTest.MovePos[5] := FxA_Exp_Pos;
		SensorTest.MovePos[6] := FxB_Exp_Pos;
		
		GroupFx.Fx_Set_A_Enc();
		
		GroupB.FindZ();
		step := step + 1;
		
	836:
		IF (GroupFx.bBuzy OR GroupFx.bError) AND (GroupB.StepA.bBuzy OR GroupB.StepA.bError) THEN
			step := step + 1;
		END_IF
		
	837:
		IF GroupFx.bDone AND GroupB.StepA.bDone THEN
			step := step + 1;
		ELSIF GroupFx.bError OR GroupB.StepA.bError THEN
			step := step + 10000;
		END_IF
		
	838:
		step := 840;
(*	===================================
				BD夾 換 AC夾
	===================================*)
	840:
		SensorTest.MovePos[7] := Sensor.sensor_test_pos;
		SensorTest.MovePos[8] := FxA_Exp_Pos;
		SensorTest.MovePos[9] := FxB_Exp_Pos;
	
		GroupFx.AC_Clamp();
		GroupFx.B_UnPress(2);
		GroupFx.D_UnPress(2);
		step := step + 1;
		
	841:
		IF (GroupFx.step_AC_C.bBuzy OR GroupFx.step_AC_C.bError) AND
			(GroupFx.step_B_P.bBuzy OR GroupFx.step_B_P.bError) AND
			 (GroupFx.step_D_P.bBuzy OR GroupFx.step_D_P.bError) THEN
			step := step + 1;
		END_IF
		
	842:
		IF GroupFx.step_AC_C.bDone AND GroupFx.step_B_P.bDone AND GroupFx.step_D_P.bDone  THEN
			step := step + 1;
		ELSIF GroupFx.step_AC_C.bError OR GroupFx.step_B_P.bError OR GroupFx.step_D_P.bError THEN
			step := step + 10000;
		END_IF
		
	843:
		tmr01.PT := T#1S;
		tmr01.IN := TRUE;
		IF tmr01.Q THEN
			tmr01.IN := FALSE;
			step := step + 1;
		END_IF
		
	844:
		SensorTest.MovePos[10] := Sensor.sensor_test_pos;
		SensorTest.MovePos[11] := FxA_Exp_Pos;
		SensorTest.MovePos[12] := FxB_Exp_Pos;
	
		GroupFx.BD_UnClamp(20);
		GroupFx.A_Press();
		GroupFx.C_Press();
		step := step + 1;
		
	845:
		IF (GroupFx.step_BD_C.bBuzy OR GroupFx.step_BD_C.bError) AND
			(GroupFx.step_A_P.bBuzy OR GroupFx.step_A_P.bError) AND
			 (GroupFx.step_C_P.bBuzy OR GroupFx.step_C_P.bError)  THEN
			step := step + 1;
		END_IF
		
	846:
		IF GroupFx.step_BD_C.bDone  THEN
// 			GroupFx.B_Press();
// 			GroupFx.D_Press();
			step := step + 1;
		ELSIF GroupFx.step_BD_C.bError THEN
			step := step + 10000;
		END_IF
		
	847:
		step := 849;
		
// 	847:
// 		IF (GroupFx.step_B_P.bBuzy OR GroupFx.step_B_P.bError) AND
// 			 (GroupFx.step_D_P.bBuzy OR GroupFx.step_D_P.bError)  THEN
// 			step := step + 1;
// 		END_IF
// 		
// 	848:
// 		IF GroupFx.step_BD_C.bDone AND GroupFx.step_A_P.bDone AND GroupFx.step_B_P.bDone AND GroupFx.step_C_P.bDone AND GroupFx.step_D_P.bDone THEN
// 			step := step + 1;
// 		ELSIF GroupFx.step_BD_C.bError OR GroupFx.step_A_P.bError OR GroupFx.step_B_P.bError OR GroupFx.step_C_P.bError OR GroupFx.step_D_P.bError THEN
// 			step := step + 10000;
// 		END_IF
	
		
	849:
		step := 850;
(*	===================================
				Fx 前往 X工作點
	===================================*)
	850:
		SensorTest.MovePos[13] := Sensor.sensor_test_pos;
		SensorTest.MovePos[14] := FxA_Exp_Pos;
		SensorTest.MovePos[15] := FxB_Exp_Pos;
		
		// BH有接縫工件
		IF ProjectData.Joint_Pos > 0 THEN
			IF Last_Pos + 1300 > ProjectData.Joint_Pos AND Fx_Exp_Pos + 1100 < ProjectData.Joint_Pos THEN
				step := step + 1;
			ELSE
				step := 855;
			END_IF
		ELSE
			step := 855;
		END_IF
	
	851:
		GroupFx.Fx_Move(ProjectData.Joint_Pos - 1400);
		step := step + 1;
		
	852:
		IF (GroupFx.bBuzy OR GroupFx.bError) THEN
			step := step + 1;
		END_IF
		
		
	853:
		IF GroupFx.bDone THEN
			step := step + 1;
		ELSIF GroupFx.bError THEN
			step := step + 10000;
		END_IF
		
	854:
		IF GroupFx.Fx_Sync_EncA_2_EncB() THEN
			step := 855;
		END_IF
		
	855:
		SensorTest.MovePos[17] := Sensor.sensor_test_pos;
		SensorTest.MovePos[18] := FxA_Exp_Pos;
		SensorTest.MovePos[19] := FxB_Exp_Pos;
		
		GroupFx.Fx_Move(Last_Pos);
		step := step + 1;
		
	856:
		IF (GroupFx.bBuzy OR GroupFx.bError) THEN
			step := step + 1;
		END_IF
		
		
	857:
		IF GroupFx.bDone THEN
			step := step + 1;
		ELSIF GroupFx.bError THEN
			step := step + 10000;
		END_IF
		
	858:
		step := 870;
		
	
		
(*	===================================
		Fx 定位後，各組測高開始
	===================================*)
	860:
		IF ProjectData.Now_Steel_Payload_A_DataNumber > 0 AND Sensor.sensorA.fDistance > 0 THEN
			GroupA.FindZ();
		END_IF
		IF ProjectData.Now_Steel_Payload_B_DataNumber > 0 AND Sensor.sensorB.fDistance > 0 THEN
			GroupB.FindZ();
		END_IF
		IF ProjectData.Now_Steel_Payload_C_DataNumber > 0 AND Sensor.sensorC.fDistance > 0 THEN
			GroupC.FindZ();
		END_IF
		IF ProjectData.Now_Steel_Payload_D_DataNumber > 0 AND Sensor.sensorD.fDistance > 0 THEN
			GroupD.FindZ();
		END_IF
		step := step + 1;
		
	861:
		IF (GroupA.StepA.bBuzy OR GroupA.StepA.bError OR ProjectData.Now_Steel_Payload_A_DataNumber = 0 OR Sensor.sensorA.fDistance = 0) AND
			(GroupB.StepA.bBuzy OR GroupB.StepA.bError OR ProjectData.Now_Steel_Payload_B_DataNumber = 0 OR Sensor.sensorB.fDistance = 0) AND
			(GroupC.StepA.bBuzy OR GroupC.StepA.bError OR ProjectData.Now_Steel_Payload_C_DataNumber = 0 OR Sensor.sensorC.fDistance = 0) AND
			(GroupD.StepA.bBuzy OR GroupD.StepA.bError OR ProjectData.Now_Steel_Payload_D_DataNumber = 0 OR Sensor.sensorD.fDistance = 0) THEN
				step := step + 1;
		END_IF
		
	862:
		GroupA.ReadyToMove := (GroupA.StepA.bDone OR Sensor.sensorA.fDistance = 0);
		GroupB.ReadyToMove := (GroupB.StepA.bDone OR Sensor.sensorB.fDistance = 0);
		GroupC.ReadyToMove := (GroupC.StepA.bDone OR Sensor.sensorC.fDistance = 0);
		GroupD.ReadyToMove := (GroupD.StepA.bDone OR Sensor.sensorD.fDistance = 0);
		IF (GroupA.StepA.bDone OR ProjectData.Now_Steel_Payload_A_DataNumber = 0 OR Sensor.sensorA.fDistance = 0) AND
			(GroupB.StepA.bDone OR ProjectData.Now_Steel_Payload_B_DataNumber = 0 OR Sensor.sensorB.fDistance = 0) AND
			(GroupC.StepA.bDone OR ProjectData.Now_Steel_Payload_C_DataNumber = 0 OR Sensor.sensorC.fDistance = 0) AND 
			(GroupD.StepA.bDone OR ProjectData.Now_Steel_Payload_D_DataNumber = 0 OR Sensor.sensorD.fDistance = 0) THEN
			 	step := step + 1;
		ELSIF 
			(GroupA.StepA.bError AND ProjectData.Now_Steel_Payload_A_DataNumber > 0) OR
			(GroupB.StepA.bError AND ProjectData.Now_Steel_Payload_B_DataNumber > 0) OR 
			(GroupC.StepA.bError AND ProjectData.Now_Steel_Payload_C_DataNumber > 0) OR 
			(GroupD.StepA.bError AND ProjectData.Now_Steel_Payload_D_DataNumber > 0) THEN
				step := step + 10000;
		END_IF
		
	863:
		step := 870;
		
(*	=============================================
				開始各組區域打標
	=============================================*)
	870: 
		tmr01.PT := T#0.5S;
		tmr01.IN := TRUE;
		IF tmr01.Q THEN
			tmr01.IN := FALSE;
			step := step + 1;
		END_IF
		
	871:
		GroupA.ReadyToMove := TRUE;
		GroupB.ReadyToMove := TRUE;
		GroupC.ReadyToMove := TRUE;
		GroupD.ReadyToMove := TRUE;
		GroupA.ReadyToPrint := TRUE;
		GroupB.ReadyToPrint := TRUE;
		GroupC.ReadyToPrint := TRUE;
		GroupD.ReadyToPrint := TRUE;
		step := step + 1;
		
	872:
		IF GroupA.bDone AND GroupB.bDone AND GroupC.bDone AND GroupD.bDone THEN
			step := step + 1;
		ELSIF GroupA.bError OR GroupB.bError OR GroupC.bError OR GroupD.bError THEN
			step := step + 10000;
		END_IF
		
	873:
		step := 880;
		
	
	880:
		step := 800;
		
END_CASE
END_ACTION

ACTION step_0900_AutoMode_GoPrintPoint_Cycle_200_Down:
(*=====================================
				搜尋 X工作點
=======================================*)

CASE step OF
(*	===================================
				搜尋 X工作點
	===================================*)
	900:
		sql_hand := ReadSQLData.Get_X_NextPos(Last_Pos);
		IF sql_hand <> 0 THEN
			step := step + 1;
		END_IF
		
	901:
		IF ReadSQLData.bBuzy OR ReadSQLData.bError THEN
			step := step + 1;
		END_IF
		
	902:
		IF ReadSQLData.bDone = sql_hand THEN
			step := step + 1;
		ELSIF ReadSQLData.bError THEN
			step := step + 10000;
		END_IF
		
	903:
		Last_Pos := ReadSQLData.fNext_XPos;
		
		// ============ 紀錄啟動條件 ============
		_log.fbJson.StartObject();
		_log.fbJson.AddKeyString('StepName','Get_Next_XPos');
		_log.fbJson.AddKeyLreal('fNext_XPos', Last_Pos);
		_log.JsonOutput();
		// ======================================
		
		_debug_X_NextPos[_debug_X_NextPos_count] := Last_Pos;
		_debug_X_NextPos_count := _debug_X_NextPos_count + 1;
		
		step := step + 1;
		
	904:
		IF Last_Pos = -1 THEN
			step := 906;
		ELSE
			step := step + 1;
		END_IF
		
	905:
		step := 910;
		
	906:
		GroupB.ToStanby(Speed:= SpdC.HighSpeed);
		step := step + 1;
		
	907:
		IF GroupB.StepA.bBuzy OR GroupB.StepA.bError THEN
			step := step + 1;
		END_IF
		
	908:
		IF GroupB.StepA.bDone THEN
			step := step + 1;
		ELSIF GroupB.StepA.bError THEN
			step := step + 10000;
		END_IF
		
	909:
		step := 1000;
		
(*	==========================================
				取得區間的打標工作
	==========================================*)
	910:
		sql_hand := ReadSQLData.Get_Payload(Start_Pos := Last_Pos, End_Pos := Last_Pos + 1);
		IF sql_hand <> 0 THEN
			step := step + 1;
		END_IF
		
	911:
		IF ReadSQLData.bBuzy OR ReadSQLData.bError THEN
			step := step + 1;
		END_IF
		
	912:
		IF ReadSQLData.bDone = sql_hand THEN
			step := step + 1;
		ELSIF ReadSQLData.bError THEN
			step := step + 10000;
		END_IF
		
	913:
		step := 920;

(*	==========================================
			設定各軸組 並 預移到打標點
	==========================================*)
	920: // 設定 各軸組 X參考座標
		GroupA.Set_X_Ref(Value := Last_Pos);
		GroupB.Set_X_Ref(Value := Last_Pos);
		GroupC.Set_X_Ref(Value := Last_Pos);
		GroupD.Set_X_Ref(Value := Last_Pos);
		step := step + 1;
		
	921:
		GroupA.ReadyToPrint := FALSE;
		GroupB.ReadyToPrint := FALSE;
		GroupC.ReadyToPrint := FALSE;
		GroupD.ReadyToPrint := FALSE;
		
		GroupA.ReadyToMove := FALSE;
		GroupB.ReadyToMove := FALSE;
		GroupC.ReadyToMove := FALSE;
		GroupD.ReadyToMove := FALSE;
		step := step + 1;
		

	
	922: // 載入區域工作內容 + 預移動開始
		GroupA.Do_WorkList();
		GroupB.Do_WorkList();
		GroupC.Do_WorkList();
		GroupD.Do_WorkList();
		step := step + 1;
		
	923:
		IF (GroupA.bBuzy OR GroupA.bError OR ProjectData.Now_Steel_Payload_A_DataNumber = 0) AND
			(GroupB.bBuzy OR GroupB.bError OR ProjectData.Now_Steel_Payload_B_DataNumber = 0) AND
			(GroupC.bBuzy OR GroupC.bError OR ProjectData.Now_Steel_Payload_C_DataNumber = 0) AND
			(GroupD.bBuzy OR GroupD.bError OR ProjectData.Now_Steel_Payload_D_DataNumber = 0) THEN
				step := step + 1;
		END_IF
		
	924:
		step := 930;
		
(*	===================================
			判斷是否走快到結尾
			如果是則交換編碼器
	===================================*)
	930: // 判斷是否走快到結尾
		IF (Last_Pos + 1100) > ProjectData.Now_Steel.Length AND GroupFx.b_BD_Clamp THEN
			IF Fx.fPos < 1000 THEN
				// 料還沒到 前端
				step := step + 1;
			ELSE
				// 料已超過 前端
				step := 935;
			END_IF
		ELSE
			step := 950;
		END_IF
		
		
	931:
		SensorTest.MovePos[0] := Sensor.sensor_test_pos;
		SensorTest.MovePos[1] := FxA_Exp_Pos;
		SensorTest.MovePos[2] := FxB_Exp_Pos;
		
		GroupFx.Fx_Move(1000);
		step := step + 1;
		
	932:
		IF (GroupFx.bBuzy OR GroupFx.bError) THEN
			step := step + 1;
		END_IF
		
		
	933:
		IF GroupFx.bDone THEN
			step := step + 1;
		ELSIF GroupFx.bError THEN
			step := step + 10000;
		END_IF
		
	934:
		step := 935;
		
	935:
		SensorTest.MovePos[4] := Sensor.sensor_test_pos;
		SensorTest.MovePos[5] := FxA_Exp_Pos;
		SensorTest.MovePos[6] := FxB_Exp_Pos;
		
		GroupFx.Fx_Set_A_Enc();
		GroupB.ToStanby(Speed:= SpdC.HighSpeed);
		step := step + 1;
		
	936:
		IF (GroupFx.bBuzy OR GroupFx.bError) AND 
			(GroupB.StepA.bBuzy OR GroupB.StepA.bError) THEN
			step := step + 1;
		END_IF
		
	937:
		IF GroupFx.bDone AND GroupB.StepA.bDone THEN
			step := step + 1;
		ELSIF GroupFx.bError OR GroupB.StepA.bError THEN
			step := step + 10000;
		END_IF
		
	938:
		step := 940;
(*	===================================
				BD夾 換 AC夾
	===================================*)
	940:
		SensorTest.MovePos[7] := Sensor.sensor_test_pos;
		SensorTest.MovePos[8] := FxA_Exp_Pos;
		SensorTest.MovePos[9] := FxB_Exp_Pos;
	
		GroupFx.AC_Clamp();
		GroupFx.B_UnPress(2);
		GroupFx.D_UnPress(2);
		step := step + 1;
		
	941:
		IF (GroupFx.step_AC_C.bBuzy OR GroupFx.step_AC_C.bError) AND
			(GroupFx.step_B_P.bBuzy OR GroupFx.step_B_P.bError) AND
			 (GroupFx.step_D_P.bBuzy OR GroupFx.step_D_P.bError) THEN
			step := step + 1;
		END_IF
		
	942:
		IF GroupFx.step_AC_C.bDone AND GroupFx.step_B_P.bDone AND GroupFx.step_D_P.bDone  THEN
			step := step + 1;
		ELSIF GroupFx.step_AC_C.bError OR GroupFx.step_B_P.bError OR GroupFx.step_D_P.bError THEN
			step := step + 10000;
		END_IF
		
	943:
		tmr01.PT := T#1S;
		tmr01.IN := TRUE;
		IF tmr01.Q THEN
			tmr01.IN := FALSE;
			step := step + 1;
		END_IF
		
	944:
		SensorTest.MovePos[10] := Sensor.sensor_test_pos;
		SensorTest.MovePos[11] := FxA_Exp_Pos;
		SensorTest.MovePos[12] := FxB_Exp_Pos;
	
		GroupFx.BD_UnClamp(20);
		GroupFx.A_Press();
		GroupFx.C_Press();
		step := step + 1;
		
	945:
		IF (GroupFx.step_BD_C.bBuzy OR GroupFx.step_BD_C.bError) AND
			(GroupFx.step_A_P.bBuzy OR GroupFx.step_A_P.bError) AND
			 (GroupFx.step_C_P.bBuzy OR GroupFx.step_C_P.bError)  THEN
			step := step + 1;
		END_IF
		
	946:
		IF GroupFx.step_BD_C.bDone THEN
// 			GroupFx.B_Press();
// 			GroupFx.D_Press();
			step := step + 1;
		ELSIF GroupFx.step_BD_C.bError THEN
			step := step + 10000;
		END_IF
		
	947:
		step := 949;
		
// 	947:
// 		IF (GroupFx.step_B_P.bBuzy OR GroupFx.step_B_P.bError) AND (GroupFx.step_D_P.bBuzy OR GroupFx.step_D_P.bError)  THEN
// 			step := step + 1;
// 		END_IF
// 		
// 	948:
// 		IF GroupFx.step_A_P.bDone AND GroupFx.step_B_P.bDone AND GroupFx.step_C_P.bDone AND GroupFx.step_D_P.bDone THEN
// 			step := step + 1;
// 		ELSIF GroupFx.step_A_P.bError OR GroupFx.step_B_P.bError OR GroupFx.step_C_P.bError OR GroupFx.step_D_P.bError THEN
// 			step := step + 10000;
// 		END_IF
		
	949:
		step := 950;
		
	950:
		GbZ.AbsMove(GroupB_Now_Z, spdc.HomeSpeed);
		step := step + 1;
		
	951:
		IF (GbZ.bBuzy OR GbZ.bError)  THEN
			step := step + 1;
		END_IF
		
	952:
		step := 970;
(*	===================================
				Fx 前往 X工作點
	===================================*)
	970:
		SensorTest.MovePos[13] := Sensor.sensor_test_pos;
		SensorTest.MovePos[14] := FxA_Exp_Pos;
		SensorTest.MovePos[15] := FxB_Exp_Pos;
		
		GroupFx.Fx_Move(Last_Pos);
		step := step + 1;
		
	971:
		IF (GroupFx.bBuzy OR GroupFx.bError) THEN
			step := step + 1;
		END_IF
		
		
	972:
		IF GroupFx.bDone AND GbZ.bDone THEN
			step := step + 1;
		ELSIF GroupFx.bError AND GbZ.bError THEN
			step := step + 10000;
		END_IF
		
	973:
		SensorTest.MovePos[17] := Sensor.sensor_test_pos;
		SensorTest.MovePos[18] := FxA_Exp_Pos;
		SensorTest.MovePos[19] := FxB_Exp_Pos;
		step := 980;
		
(*	===================================
		原測高動作，小隻的料不做
	===================================*)

		
(*	=============================================
				開始各組區域打標
	=============================================*)
	980: 
		tmr01.PT := T#1S;
		tmr01.IN := TRUE;
		IF tmr01.Q THEN
			tmr01.IN := FALSE;
			step := step + 1;
		END_IF
		
	981:
		GroupA.ReadyToMove := TRUE;
		GroupB.ReadyToMove := TRUE;
		GroupC.ReadyToMove := TRUE;
		GroupD.ReadyToMove := TRUE;
		GroupA.ReadyToPrint := TRUE;
		GroupB.ReadyToPrint := TRUE;
		GroupC.ReadyToPrint := TRUE;
		GroupD.ReadyToPrint := TRUE;
		step := step + 1;
		
	982:
		IF GroupA.bDone AND GroupB.bDone AND GroupC.bDone AND GroupD.bDone THEN
			step := step + 1;
		ELSIF GroupA.bError OR GroupB.bError OR GroupC.bError OR GroupD.bError THEN
			step := step + 10000;
		END_IF
		
	983:
		step := 990;
		
	
	990:
		step := 900;
		
END_CASE
END_ACTION

ACTION step_1000_AutoPrgEnd:
CASE step OF
	1000:
		uRunCounter := uRunCounter + 1;
		ProjectData.old_Steel := ProjectData.Now_Steel;
		GroupA.Oil();
		GroupB.Oil();
		GroupC.Oil();
		GroupD.Oil();
		step := step + 1;
		
	1001:
		sql_hand := ReadSQLData.Set_Steel_Finish(uid := ProjectData.Now_Steel.uid);
		IF sql_hand <> 0 THEN
			step := step + 1;
		END_IF
		
	1002:
		IF ReadSQLData.bBuzy OR ReadSQLData.bError THEN
			step := step + 1;
		END_IF
		
	1003:
		IF ReadSQLData.bDone = sql_hand OR ReadSQLData.bError THEN
			ProjectData.WorkOrder_Now.steel_id := '';
			step := step + 1;
		END_IF
		
	1004:
		step := 1010;
		

	1010:
		sql_hand := ReadSQLData.Get_Steel_Num_On_Wait();
		IF sql_hand <> 0 THEN
			step := step + 1;
		END_IF
		
	1011:
		GroupA.ToStanby(spdc.HighSpeed);
		GroupB.ToStanby(spdc.HighSpeed);
		GroupC.ToStanby(spdc.HighSpeed);
		GroupD.ToStanby(spdc.HighSpeed);
		GroupFx.A_UnPress(5);
		GroupFx.B_UnPress(5);
		GroupFx.C_UnPress(5);
		GroupFx.D_UnPress(5);
		IF (fx.fPos < 1800) THEN
			GroupFx.Fx_Move(1800);
		ELSE
			fx.Stop();
		END_IF
		
		step := step + 1;
		
	1012:
		IF (GroupA.StepA.bBuzy OR GroupA.StepA.bError) AND 
			(GroupB.StepA.bBuzy OR GroupB.StepA.bError) AND
			(GroupC.StepA.bBuzy OR GroupC.StepA.bError) AND
			(GroupD.StepA.bBuzy OR GroupD.StepA.bError) AND
			(GroupFx.bBuzy OR GroupFx.bError OR fx.fPos >= 1800) THEN
				step := step + 1;
		END_IF
		
	1013:
		IF (GroupFx.bDone OR fx.fPos >= 1800) THEN
			step := step + 1;
		ELSIF GroupA.StepA.bError OR GroupB.StepA.bError OR GroupC.StepA.bError OR GroupD.StepA.bError OR GroupFx.bError THEN
			step := step + 10000;
		END_IF
		
	1014:
		
		step := 1020;
		
	1020:
// 		GroupFx.A_UnPress(5);
// 		GroupFx.B_UnPress(5);
// 		GroupFx.C_UnPress(5);
// 		GroupFx.D_UnPress(5);
		step := step + 1;
		
	1021:
		step := step + 1;
// 		IF (GroupFx.step_A_P.bBuzy OR GroupFx.step_A_P.bError) AND
// 			(GroupFx.step_B_P.bBuzy OR GroupFx.step_B_P.bError) AND
// 			(GroupFx.step_C_P.bBuzy OR GroupFx.step_C_P.bError) AND
// 			(GroupFx.step_D_P.bBuzy OR GroupFx.step_D_P.bError) THEN
// 				step := step + 1;
// 		END_IF
		
	1022:
		tmr01.PT:= T#2S;
		tmr01.IN := TRUE;
		IF tmr01.Q THEN
			tmr01.IN := FALSE;
			step := step + 1;
		END_IF
		
// 		IF GroupFx.step_A_P.bDone AND 
// 			GroupFx.step_B_P.bDone AND 
// 			GroupFx.step_C_P.bDone AND 
// 			GroupFx.step_D_P.bDone THEN
// 				step := step + 1;
// 		ELSIF GroupFx.step_A_P.bError AND 
// 			GroupFx.step_B_P.bError AND 
// 			GroupFx.step_C_P.bError AND 
// 			GroupFx.step_D_P.bError THEN
// 				step := step + 10000;
// 		END_IF
		
	1023:
		step := 1030;
		
		
	1030:
		GroupFx.AC_UnClamp(10);
		GroupFx.BD_UnClamp(10);
		step := step + 1;
		
	1031:
		IF (GroupFx.step_AC_C.bBuzy OR GroupFx.step_AC_C.bError) AND
			(GroupFx.step_BD_C.bBuzy OR GroupFx.step_BD_C.bError) THEN
				step := step + 1;
		END_IF
		
	1032:
		tmr01.PT := T#2S;
		tmr01.IN := TRUE;
		IF tmr01.Q THEN
			tmr01.IN := FALSE;
			step := step + 1;
		END_IF
		
	1033:
		IF ReadSQLData.bDone = sql_hand OR ReadSQLData.bError THEN
			step := 1040;
		END_IF
		
	1040:
		ExpConver.OutRollerStart();
		step := step + 1;
		
	1041:
		IF ExpConver.Out_Moter_Running THEN
			step := step + 1;
		END_IF
		
	1042:
		IF ProjectData.Now_Steel.Length < 11000 THEN
			tmr01.PT := T#2S;
		ELSE
			tmr01.PT := T#0.5S;
		END_IF
		tmr01.IN := NOT io.i709;
		IF tmr01.Q THEN
			tmr01.IN := FALSE;
			step := step + 1;
		END_IF
		
	1043:
		ExpConver.OutRollerStop();
		step := step + 1;
		
	1044:
		IF NOT ExpConver.Out_Moter_Running THEN
			step := step + 1;
		END_IF
		
	1045:
		IF ReadSQLData.bDone = sql_hand OR ReadSQLData.bError THEN
			step := step + 1;
		END_IF
		
	1046:
		sql_hand := ReadSQLData.Get_WorkkOrder();
		step := step + 1;
		
	1047:
		IF ReadSQLData.bDone = sql_hand OR ReadSQLData.bError THEN
			step := step + 1;
		END_IF
		
	1048:
		step := 1050;
		

	1050:
		IF LEN(STR:=ProjectData.WorkOrder_inSide.steel_id) > 0 THEN
			// 已經有 料的狀態 是 在輸送滾輪上(inSide)
			ProjectData.WorkOrder_Now := ProjectData.WorkOrder_inSide;
			step := 1060;
		ELSIF ProjectData.WorkOrder_Num_On_Wait > 0  THEN
			IF ExpConver.Feed_bDone THEN
				step := step + 1;
			ELSE
				step := 1054;
			END_IF
		ELSE
			step := 1090;
		END_IF
		
	1051:	
		IF NOT ExpConver.Feed_bBuzy THEN
			ExpConver.FeedAutoStart();
			Hmi_Web.Auto_Start := FALSE;
			step := step + 1;
		ELSIF (ExpConver.ActionMode_Now > 400 AND ExpConver.ActionMode_Now < 800) THEN
			step := 1060;
		END_IF
		
	1052:
		IF ExpConver.Feed_bBuzy OR ExpConver.Feed_bError OR ExpConver.ActionMode_Now = 806 THEN
			step := step + 1;
		END_IF
		
	1053:
		IF ExpConver.Feed_bDone THEN
			step := step + 1;
		ELSIF ExpConver.Feed_bError THEN
			step := step + 10000;
		END_IF
		
	1054:
		step := 1060;


(*	========================================
			讀取資料庫 取得排程資料
	========================================*)
	1060:
		IF NOT ExpConver.Feed_bBuzy OR (ExpConver.ActionMode_Now > 400 AND ExpConver.ActionMode_Now < 800) THEN
			step := step + 1;
		END_IF
		
	1061:	
		sql_hand := ReadSQLData.Get_WorkkOrder();
		IF sql_hand <> 0 THEN
			step := step + 1;
		END_IF
			
	1062:
		IF ReadSQLData.bBuzy OR ReadSQLData.bError THEN
			step := step + 1;
		END_IF
			
	1063:
		IF ReadSQLData.bDone = sql_hand THEN
			step := step + 1;
		ELSIF ReadSQLData.bError THEN
			step := step + 10000;
		END_IF
		
	1064:
		IF LEN(STR:=ProjectData.WorkOrder_inSide.steel_id) > 0 THEN
			// 已經有 料的狀態 是 在輸送滾輪上(inSide)
			ProjectData.WorkOrder_Now := ProjectData.WorkOrder_inSide;
			step := 1070;
		ELSE
			// 沒有 料的狀態 是 在輸送滾輪上(inSide)
			step := 1090;
		END_IF
		

(*	========================================
				有進料完成的料
	========================================*)
	1070:
		sql_hand := ReadSQLData.Get_SteelData(ProjectData.WorkOrder_Now.steel_id);
		IF sql_hand <> 0 THEN
			step := step + 1;
		END_IF
			
	1071:
		IF ReadSQLData.bBuzy OR ReadSQLData.bError THEN
			step := step + 1;
		END_IF
		
	1072:
		IF ReadSQLData.bDone = sql_hand THEN
			step := step + 1;
		ELSIF ReadSQLData.bError THEN
			step := step + 10000;
		END_IF
		
	1073:
		
		step := 600;
		
		
	1090:
		GroupFx.AC_UnClamp();
		GroupFx.BD_UnClamp();
		GroupFx.A_UnPress();
		GroupFx.B_UnPress();
		GroupFx.C_UnPress();
		GroupFx.D_UnPress();
		step := step + 1;
		
	1091:
		IF (GroupFx.step_AC_C.bBuzy OR GroupFx.step_AC_C.bError) AND
			(GroupFx.step_BD_C.bBuzy OR GroupFx.step_BD_C.bError) THEN
				step := step + 1;
		END_IF
		
	1092:
		tmr01.PT := T#2S;
		tmr01.IN := TRUE;
		IF tmr01.Q THEN
			tmr01.IN := FALSE;
			step := step + 1;
		END_IF
		
	1093:
		step := 0;
		
	step := 0;
END_CASE
END_ACTION

ACTION step_7000_test_mask_A:
CASE step OF
	7000:
		iCount := 1;
		fPointStart[1] := GaX.Pos;
		fPointStart[2] := GaY.Pos;
		step := 7010;
		
	7010:// 載入DXF專案
		LaserMark.laserA.Load_Project('test');
		step := step + 1;
		
	7011:
		IF LaserMark.laserA.bBuzy OR LaserMark.laserA.bError THEN
			step := step + 1;
		END_IF
		
	7012:
		IF LaserMark.laserA.bDone THEN
			step := step + 1;
		ELSIF LaserMark.laserA.bError THEN
			step := step + 10000;
		END_IF
		
	7013:
		step := 7020;
		
	7020: // 移X軸
		GaX.RelMove(80,80);
// 		GaX.RelMove(fPoint[iCount,1],80);
// 		GaY.RelMove(fPoint[iCount,2],80);
// 		LaserMark.laserA.Edit_Object(name := 'dxf', Content := sFilename[iCount]);
		step := step + 1;
		
	7021:
// 		IF (GaX.bBuzy OR GaX.bError) AND (GaY.bBuzy OR GaY.bError) AND (LaserMark.laserA.bBuzy OR LaserMark.laserA.bError) THEN
// 			step := step + 1;
// 		END_IF
		IF (GaX.bBuzy OR GaX.bError) THEN
			step := step + 1;
		END_IF
		
	7022:
		IF GaX.bDone THEN
			step := step + 1;
		ELSIF GaX.bError THEN
			step := step + 10000;
		END_IF
		
	7023:
		step := 7030;
		
	7030: // 換置 DXF檔案
// 		step := step + 1;
		step := 7035;
		
// 	7031:
// 		IF LaserMark.laserA.bDone THEN
// 			step := step + 1;
// 		ELSIF LaserMark.laserA.bError THEN
// 			step := step + 10000;
// 		END_IF
// 		
// 	7032:
// 		tmr01.IN := TRUE;
// 		tmr01.PT := T#500MS;
// 		IF tmr01.Q THEN
// 			tmr01.IN := FALSE;
// 			step := step + 1;
// 		END_IF
// 		
// 	7033:
// 		step := 7035;
		
		
	7035: // 打雷射
		LaserMark.laserA.Mark();
		step := step + 1;
		
	7036:
		IF LaserMark.laserA.bBuzy OR LaserMark.laserA.bError THEN
			step := step + 1;
		END_IF
		
	7037:
		IF LaserMark.laserA.bDone THEN
			step := step + 1;
		ELSIF LaserMark.laserA.bError THEN
			step := step + 10000;
		END_IF
		
	7038:
		tmr01.PT := T#500MS;
		tmr01.IN := TRUE;
		IF tmr01.Q THEN
			tmr01.IN := FALSE;
			step := step + 1;
		END_IF
		
	7039:
		step := 7040;
		
	7040:
		IF iCount < 4 THEN
			iCount := iCount + 1;
			step := 7020;
		ELSE
			iCount := 1;
			step := step + 1;
		END_IF
		
	7041:
		GaX.AbsMove(fPointStart[1],80);
		GaY.AbsMove(fPointStart[2],80);
		step := step + 1;
		
	7042:
		IF (GaX.bBuzy OR GaX.bError) AND (GaY.bBuzy OR GaY.bError) THEN
			step := step + 1;
		END_IF
		
	7043:
		IF GaX.bDone AND GaY.bDone THEN
			step := step + 1;
		ELSIF GaX.bError OR GaY.bError THEN
			step := step + 10000;
		END_IF
		
	7044:
		step := 0;
END_CASE
END_ACTION

ACTION step_7100_test_mask_A_1:

CASE step OF
	7100:
		iCount := 1;
		fPointStart[1] := GaX.Pos;
		fPointStart[2] := GaY.Pos;
		step := step + 1;
		
	7101:
		GroupA.FindZ_Fast();
		step := step + 1;
		
	7102:
		IF (GroupA.StepA.bBuzy OR GroupA.StepA.bError) THEN
			step := step + 1;
		END_IF
		
	7103:
		IF GroupA.StepA.bDone THEN
			step := step + 1;
		ELSIF GroupA.StepA.bError THEN
			step := step + 10000;
		END_IF
		
	7104:
		step := 7120;
		
	7120: // 移X軸
		GaX.RelMove(fPoint2[iCount,1],80);
		GaY.RelMove(fPoint2[iCount,2],80);
		step := step + 1;
		
	7121:
		IF (GaX.bBuzy OR GaX.bError) AND (GaY.bBuzy OR GaY.bError) THEN
			step := step + 1;
		END_IF
		
	7122:
		IF GaX.bDone AND GaY.bDone THEN
			step := step + 1;
		ELSIF GaX.bError OR GaY.bError THEN
			step := step + 10000;
		END_IF
		
	7123:
		step := 7130;
		
		
	7130: // 打雷射
		LaserMark.laserA.Mark();
		step := step + 1;
		
	7131:
		IF LaserMark.laserA.bBuzy OR LaserMark.laserA.bError THEN
			step := step + 1;
		END_IF
		
	7132:
		IF LaserMark.laserA.bDone THEN
			step := step + 1;
		ELSIF LaserMark.laserA.bError THEN
			step := step + 10000;
		END_IF
		
	7133:
		tmr01.PT := T#500MS;
		tmr01.IN := TRUE;
		IF tmr01.Q THEN
			tmr01.IN := FALSE;
			step := step + 1;
		END_IF
		
	7134:
		step := 7140;
		
	7140:
		IF iCount < 4 THEN
			iCount := iCount + 1;
			step := 7120;
		ELSE
			iCount := iCount + 1;
			step := step + 1;
		END_IF
		
	7141:
		GaX.AbsMove(fPointStart[1] + 5,80);
		GaY.AbsMove(fPointStart[2] + 5,80);
		step := step + 1;
		
	7142:
		IF (GaX.bBuzy OR GaX.bError) AND (GaY.bBuzy OR GaY.bError) THEN
			step := step + 1;
		END_IF
		
	7143:
		IF GaX.bDone AND GaY.bDone THEN
			step := step + 1;
		ELSIF GaX.bError OR GaY.bError THEN
			step := step + 10000;
		END_IF
		
	7144:
		iCount := 0;
		step := 0;
END_CASE
END_ACTION

ACTION step_7200_test_mask_B:
CASE step OF
	7000:
		iCount := 1;
		fPointStart[1] := GaX.Pos;
		fPointStart[2] := GaY.Pos;
		step := 7010;
		
	7010:// 載入DXF專案
		LaserMark.laserA.Load_Project('dxf');
		step := step + 1;
		
	7011:
		IF LaserMark.laserA.bBuzy OR LaserMark.laserA.bError THEN
			step := step + 1;
		END_IF
		
	7012:
		IF LaserMark.laserA.bDone THEN
			step := step + 1;
		ELSIF LaserMark.laserA.bError THEN
			step := step + 10000;
		END_IF
		
	7013:
		step := 7020;
		
	7020: // 移X軸
		GaX.RelMove(fPoint[iCount,1],80);
		GaY.RelMove(fPoint[iCount,2],80);
		LaserMark.laserA.Edit_Object(Name := 'dxf', Content := sFilename[iCount]);
		step := step + 1;
		
	7021:
		IF (GaX.bBuzy OR GaX.bError) AND (GaY.bBuzy OR GaY.bError) AND (LaserMark.laserA.bBuzy OR LaserMark.laserA.bError) THEN
			step := step + 1;
		END_IF
		
	7022:
		IF GaX.bDone AND GaY.bDone THEN
			step := step + 1;
		ELSIF GaX.bError OR GaY.bError THEN
			step := step + 10000;
		END_IF
		
	7023:
		step := 7030;
		
	7030: // 換置 DXF檔案
		step := step + 1;
		
	7031:
		IF LaserMark.laserA.bDone THEN
			step := step + 1;
		ELSIF LaserMark.laserA.bError THEN
			step := step + 10000;
		END_IF
		
	7032:
		tmr01.IN := TRUE;
		tmr01.PT := T#500MS;
		IF tmr01.Q THEN
			tmr01.IN := FALSE;
			step := 7035;
		END_IF
		
		
	7035: // 打雷射
		LaserMark.laserA.Mark();
		step := step + 1;
		
	7036:
		IF LaserMark.laserA.bBuzy OR LaserMark.laserA.bError THEN
			step := step + 1;
		END_IF
		
	7037:
		IF LaserMark.laserA.bDone THEN
			step := step + 1;
		ELSIF LaserMark.laserA.bError THEN
			step := step + 10000;
		END_IF
		
	7038:
		tmr01.PT := T#500MS;
		tmr01.IN := TRUE;
		IF tmr01.Q THEN
			tmr01.IN := FALSE;
			step := step + 1;
		END_IF
		
	7039:
		step := 7040;
		
	7040:
		IF iCount < 9 THEN
			iCount := iCount + 1;
			step := 7020;
		ELSE
			iCount := 1;
			step := step + 1;
		END_IF
		
	7041:
		GaX.AbsMove(fPointStart[1],80);
		GaY.AbsMove(fPointStart[2],80);
		step := step + 1;
		
	7042:
		IF (GaX.bBuzy OR GaX.bError) AND (GaY.bBuzy OR GaY.bError) THEN
			step := step + 1;
		END_IF
		
	7043:
		IF GaX.bDone AND GaY.bDone THEN
			step := step + 1;
		ELSIF GaX.bError OR GaY.bError THEN
			step := step + 10000;
		END_IF
		
	7044:
		step := 0;
END_CASE
END_ACTION

ACTION step_7300_test_mask_B_1:

CASE step OF
	7200:
		iCount := 1;
		fPointStart[1] := GaX.Pos;
		fPointStart[2] := GaY.Pos;
		step := 7220;
		
	7220: // 移X軸
		GaX.RelMove(fPoint2[iCount,1],80);
		GaY.RelMove(fPoint2[iCount,2],80);
		step := step + 1;
		
	7221:
		IF (GaX.bBuzy OR GaX.bError) AND (GaY.bBuzy OR GaY.bError) THEN
			step := step + 1;
		END_IF
		
	7222:
		IF GaX.bDone AND GaY.bDone THEN
			step := step + 1;
		ELSIF GaX.bError OR GaY.bError THEN
			step := step + 10000;
		END_IF
		
	7223:
		step := 7230;
		
		
	7230: // 打雷射
		LaserMark.laserA.Mark();
		step := step + 1;
		
	7231:
		IF LaserMark.laserA.bBuzy OR LaserMark.laserA.bError THEN
			step := step + 1;
		END_IF
		
	7232:
		IF LaserMark.laserA.bDone THEN
			step := step + 1;
		ELSIF LaserMark.laserA.bError THEN
			step := step + 10000;
		END_IF
		
	7233:
		tmr01.PT := T#500MS;
		tmr01.IN := TRUE;
		IF tmr01.Q THEN
			tmr01.IN := FALSE;
			step := step + 1;
		END_IF
		
	7234:
		step := 7240;
		
	7240:
		IF iCount < 4 THEN
			iCount := iCount + 1;
			step := 7220;
		ELSE
			
			iCount := iCount + 1;
			step := step + 1;
		END_IF
		
	7241:
		GaX.AbsMove(fPointStart[1],80);
		GaY.AbsMove(fPointStart[2],80);
		step := step + 1;
		
	7242:
		IF (GaX.bBuzy OR GaX.bError) AND (GaY.bBuzy OR GaY.bError) THEN
			step := step + 1;
		END_IF
		
	7243:
		IF GaX.bDone AND GaY.bDone THEN
			step := step + 1;
		ELSIF GaX.bError OR GaY.bError THEN
			step := step + 10000;
		END_IF
		
	7244:
		iCount := 0;
		step := 0;

		
END_CASE
END_ACTION

ACTION step_7400_test_mask_C:
CASE step OF
	7400:
		iCount := 1;
		fPointStart[1] := GcX.Pos;
		fPointStart[2] := GcY.Pos;
		step := 7410;
		
	7410:// 載入DXF專案
		LaserMark.laserC.Load_Project('dxf');
		step := step + 1;
		
	7411:
		IF LaserMark.laserC.bBuzy OR LaserMark.laserC.bError THEN
			step := step + 1;
		END_IF
		
	7412:
		IF LaserMark.laserC.bDone THEN
			step := step + 1;
		ELSIF LaserMark.laserC.bError THEN
			step := step + 10000;
		END_IF
		
	7413:
		step := 7420;
		
	7420: // 移X軸
		GcX.RelMove(fPoint[iCount,1],80);
		GcY.RelMove(fPoint[iCount,2],80);
		LaserMark.laserC.Edit_Object(Name := 'dxf', Content := sFilename[iCount]);
		step := step + 1;
		
	7421:
		IF (GcX.bBuzy OR GcX.bError) AND (GcY.bBuzy OR GcY.bError) AND (LaserMark.laserC.bBuzy OR LaserMark.laserC.bError) THEN
			step := step + 1;
		END_IF
		
	7422:
		IF GcX.bDone AND GcY.bDone THEN
			step := step + 1;
		ELSIF GcX.bError OR GcY.bError THEN
			step := step + 10000;
		END_IF
		
	7423:
		step := 7430;
		
	7430: // 換置 DXF檔案
		step := step + 1;
		
	7431:
		IF LaserMark.laserC.bDone THEN
			step := step + 1;
		ELSIF LaserMark.laserC.bError THEN
			step := step + 10000;
		END_IF
		
	7432:
		tmr01.IN := TRUE;
		tmr01.PT := T#500MS;
		IF tmr01.Q THEN
			tmr01.IN := FALSE;
			step := 7435;
		END_IF
		
		
	7435: // 打雷射
		LaserMark.laserC.Mark();
		step := step + 1;
		
	7436:
		IF LaserMark.laserC.bBuzy OR LaserMark.laserC.bError THEN
			step := step + 1;
		END_IF
		
	7437:
		IF LaserMark.laserC.bDone THEN
			step := step + 1;
		ELSIF LaserMark.laserC.bError THEN
			step := step + 10000;
		END_IF
		
	7438:
		tmr01.PT := T#500MS;
		tmr01.IN := TRUE;
		IF tmr01.Q THEN
			tmr01.IN := FALSE;
			step := step + 1;
		END_IF
		
	7439:
		step := 7440;
		
	7440:
		IF iCount < 9 THEN
			iCount := iCount + 1;
			step := 7420;
		ELSE
			iCount := 1;
			step := step + 1;
		END_IF
		
	7441:
		GcX.AbsMove(fPointStart[1],80);
		GcY.AbsMove(fPointStart[2],80);
		step := step + 1;
		
	7442:
		IF (GcX.bBuzy OR GcX.bError) AND (GcY.bBuzy OR GcY.bError) THEN
			step := step + 1;
		END_IF
		
	7443:
		IF GcX.bDone AND GcY.bDone THEN
			step := step + 1;
		ELSIF GcX.bError OR GcY.bError THEN
			step := step + 10000;
		END_IF
		
	7444:
		step := 0;
END_CASE
END_ACTION

ACTION step_7500_test_mask_C_1:

CASE step OF
	7500:
		iCount := 1;
		fPointStart[1] := GcX.Pos;
		fPointStart[2] := GcY.Pos;
		step := 7520;
		
	7520: // 移X軸
		GcX.RelMove(fPoint2[iCount,1],80);
		GcY.RelMove(fPoint2[iCount,2],80);
		step := step + 1;
		
	7521:
		IF (GcX.bBuzy OR GcX.bError) AND (GcY.bBuzy OR GcY.bError) THEN
			step := step + 1;
		END_IF
		
	7522:
		IF GcX.bDone AND GcY.bDone THEN
			step := step + 1;
		ELSIF GcX.bError OR GcY.bError THEN
			step := step + 10000;
		END_IF
		
	7523:
		step := 7530;
		
		
	7530: // 打雷射
		LaserMark.laserC.Mark();
		step := step + 1;
		
	7531:
		IF LaserMark.laserC.bBuzy OR LaserMark.laserC.bError THEN
			step := step + 1;
		END_IF
		
	7532:
		IF LaserMark.laserC.bDone THEN
			step := step + 1;
		ELSIF LaserMark.laserC.bError THEN
			step := step + 10000;
		END_IF
		
	7533:
		tmr01.PT := T#500MS;
		tmr01.IN := TRUE;
		IF tmr01.Q THEN
			tmr01.IN := FALSE;
			step := step + 1;
		END_IF
		
	7534:
		step := 7540;
		
	7540:
		IF iCount < 4 THEN
			iCount := iCount + 1;
			step := 7520;
		ELSE
			
			iCount := iCount + 1;
			step := step + 1;
		END_IF
		
	7541:
		GcX.AbsMove(fPointStart[1],80);
		GcY.AbsMove(fPointStart[2],80);
		step := step + 1;
		
	7542:
		IF (GcX.bBuzy OR GcX.bError) AND (GcY.bBuzy OR GcY.bError) THEN
			step := step + 1;
		END_IF
		
	7543:
		IF GcX.bDone AND GcY.bDone THEN
			step := step + 1;
		ELSIF GcX.bError OR GcY.bError THEN
			step := step + 10000;
		END_IF
		
	7544:
		iCount := 0;
		step := 8010;

		
END_CASE
END_ACTION

ACTION step_7600_test_mask_D:
CASE step OF
	7600:
		iCount := 1;
		fPointStart[1] := GdX.Pos;
		fPointStart[2] := GdY.Pos;
		step := 7610;
		
	7610:// 載入DXF專案
		LaserMark.laserD.Load_Project('dxf');
		step := step + 1;
		
	7611:
		IF LaserMark.laserD.bBuzy OR LaserMark.laserD.bError THEN
			step := step + 1;
		END_IF
		
	7612:
		IF LaserMark.laserD.bDone THEN
			step := step + 1;
		ELSIF LaserMark.laserD.bError THEN
			step := step + 10000;
		END_IF
		
	7613:
		step := 7620;
		
	7620: // 移X軸
		GdX.RelMove(fPoint[iCount,1],80);
		GdY.RelMove(fPoint[iCount,2],80);
		LaserMark.laserD.Edit_Object(Name := 'dxf', Content := sFilename[iCount]);
		step := step + 1;
		
	7621:
		IF (GdX.bBuzy OR GdX.bError) AND (GdY.bBuzy OR GdY.bError) AND (LaserMark.laserD.bBuzy OR LaserMark.laserD.bError) THEN
			step := step + 1;
		END_IF
		
	7622:
		IF GdX.bDone AND GdY.bDone THEN
			step := step + 1;
		ELSIF GdX.bError OR GdY.bError THEN
			step := step + 10000;
		END_IF
		
	7623:
		step := 7630;
		
	7630: // 換置 DXF檔案
		step := step + 1;
		
	7631:
		IF LaserMark.laserD.bDone THEN
			step := step + 1;
		ELSIF LaserMark.laserD.bError THEN
			step := step + 10000;
		END_IF
		
	7632:
		tmr01.IN := TRUE;
		tmr01.PT := T#500MS;
		IF tmr01.Q THEN
			tmr01.IN := FALSE;
			step := 7635;
		END_IF
		
		
	7635: // 打雷射
		LaserMark.laserD.Mark();
		step := step + 1;
		
	7636:
		IF LaserMark.laserD.bBuzy OR LaserMark.laserD.bError THEN
			step := step + 1;
		END_IF
		
	7637:
		IF LaserMark.laserD.bDone THEN
			step := step + 1;
		ELSIF LaserMark.laserD.bError THEN
			step := step + 10000;
		END_IF
		
	7638:
		tmr01.PT := T#500MS;
		tmr01.IN := TRUE;
		IF tmr01.Q THEN
			tmr01.IN := FALSE;
			step := step + 1;
		END_IF
		
	7639:
		step := 7640;
		
	7640:
		IF iCount < 9 THEN
			iCount := iCount + 1;
			step := 7620;
		ELSE
			iCount := 1;
			step := step + 1;
		END_IF
		
	7641:
		GdX.AbsMove(fPointStart[1],80);
		GdY.AbsMove(fPointStart[2],80);
		step := step + 1;
		
	7642:
		IF (GdX.bBuzy OR GdX.bError) AND (GdY.bBuzy OR GdY.bError) THEN
			step := step + 1;
		END_IF
		
	7643:
		IF GdX.bDone AND GdY.bDone THEN
			step := step + 1;
		ELSIF GdX.bError OR GdY.bError THEN
			step := step + 10000;
		END_IF
		
	7644:
		step := 0;
END_CASE
END_ACTION

ACTION step_7700_test_mask_D_1:
CASE step OF
	7700:
		iCount := 1;
		fPointStart[1] := GdX.Pos;
		fPointStart[2] := GdY.Pos;
		step := 7720;
		
	7720: // 移X軸
		GdX.RelMove(fPoint2[iCount,1],80);
		GdY.RelMove(fPoint2[iCount,2],80);
		step := step + 1;
		
	7721:
		IF (GdX.bBuzy OR GdX.bError) AND (GdY.bBuzy OR GdY.bError) THEN
			step := step + 1;
		END_IF
		
	7722:
		IF GdX.bDone AND GdY.bDone THEN
			step := step + 1;
		ELSIF GdX.bError OR GdY.bError THEN
			step := step + 10000;
		END_IF
		
	7723:
		step := 7730;
		
		
	7730: // 打雷射
		LaserMark.laserD.Mark();
		step := step + 1;
		
	7731:
		IF LaserMark.laserD.bBuzy OR LaserMark.laserD.bError THEN
			step := step + 1;
		END_IF
		
	7732:
		IF LaserMark.laserD.bDone THEN
			step := step + 1;
		ELSIF LaserMark.laserD.bError THEN
			step := step + 10000;
		END_IF
		
	7733:
		tmr01.PT := T#500MS;
		tmr01.IN := TRUE;
		IF tmr01.Q THEN
			tmr01.IN := FALSE;
			step := step + 1;
		END_IF
		
	7734:
		step := 7740;
		
	7740:
		IF iCount < 4 THEN
			iCount := iCount + 1;
			step := 7720;
		ELSE
			
			iCount := iCount + 1;
			step := step + 1;
		END_IF
		
	7741:
		GdX.AbsMove(fPointStart[1] - 5, 80);
		GdY.AbsMove(fPointStart[2] + 5, 80);
		step := step + 1;
		
	7742:
		IF (GdX.bBuzy OR GdX.bError) AND (GdY.bBuzy OR GdY.bError) THEN
			step := step + 1;
		END_IF
		
	7743:
		IF GdX.bDone AND GdY.bDone THEN
			step := step + 1;
		ELSIF GdX.bError OR GdY.bError THEN
			step := step + 10000;
		END_IF
		
	7744:
		iCount := 0;
		step := 8010;

		
END_CASE
END_ACTION

ACTION step_7800_FindZ:
CASE step OF
	7800: // 設定 工件大小
		ProjectData.Now_Steel.Height	:= 400;
		ProjectData.Now_Steel.Width		:= 200;
		
